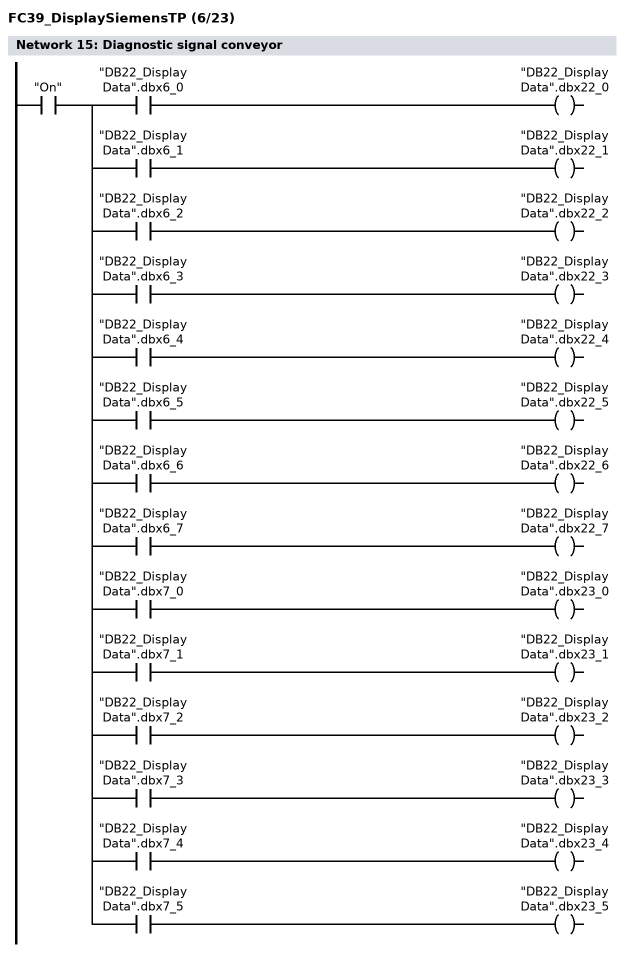
   RUNG wire#powerrail
      Contact( "On" )
      wire#w1
      Contact( "DB22_DisplayData".dbx6_0 )
      Coil( "DB22_DisplayData".dbx22_0 )
   END_RUNG
   RUNG wire#w1
      Contact( "DB22_DisplayData".dbx6_1 )
      Coil( "DB22_DisplayData".dbx22_1 )
   END_RUNG
   RUNG wire#w1
      Contact( "DB22_DisplayData".dbx6_2 )
      Coil( "DB22_DisplayData".dbx22_2 )
   END_RUNG
   RUNG wire#w1
      Contact( "DB22_DisplayData".dbx6_3 )
      Coil( "DB22_DisplayData".dbx22_3 )
   END_RUNG
   RUNG wire#w1
      Contact( "DB22_DisplayData".dbx6_4 )
      Coil( "DB22_DisplayData".dbx22_4 )
   END_RUNG
   RUNG wire#w1
      Contact( "DB22_DisplayData".dbx6_5 )
      Coil( "DB22_DisplayData".dbx22_5 )
   END_RUNG
   RUNG wire#w1
      Contact( "DB22_DisplayData".dbx6_6 )
      Coil( "DB22_DisplayData".dbx22_6 )
   END_RUNG
   RUNG wire#w1
      Contact( "DB22_DisplayData".dbx6_7 )
      Coil( "DB22_DisplayData".dbx22_7 )
   END_RUNG
   RUNG wire#w1
      Contact( "DB22_DisplayData".dbx7_0 )
      Coil( "DB22_DisplayData".dbx23_0 )
   END_RUNG
   RUNG wire#w1
      Contact( "DB22_DisplayData".dbx7_1 )
      Coil( "DB22_DisplayData".dbx23_1 )
   END_RUNG
   RUNG wire#w1
      Contact( "DB22_DisplayData".dbx7_2 )
      Coil( "DB22_DisplayData".dbx23_2 )
   END_RUNG
   RUNG wire#w1
      Contact( "DB22_DisplayData".dbx7_3 )
      Coil( "DB22_DisplayData".dbx23_3 )
   END_RUNG
   RUNG wire#w1
      Contact( "DB22_DisplayData".dbx7_4 )
      Coil( "DB22_DisplayData".dbx23_4 )
   END_RUNG
   RUNG wire#w1
      Contact( "DB22_DisplayData".dbx7_5 )
      Coil( "DB22_DisplayData".dbx23_5 )
   END_RUNG
   // the same network as SCL:
   "DB22_DisplayData".dbx22_0 := "On" AND "DB22_DisplayData".dbx6_0;
   "DB22_DisplayData".dbx22_1 := "On" AND "DB22_DisplayData".dbx6_1;
   "DB22_DisplayData".dbx22_2 := "On" AND "DB22_DisplayData".dbx6_2;
   "DB22_DisplayData".dbx22_3 := "On" AND "DB22_DisplayData".dbx6_3;
   "DB22_DisplayData".dbx22_4 := "On" AND "DB22_DisplayData".dbx6_4;
   "DB22_DisplayData".dbx22_5 := "On" AND "DB22_DisplayData".dbx6_5;
   "DB22_DisplayData".dbx22_6 := "On" AND "DB22_DisplayData".dbx6_6;
   "DB22_DisplayData".dbx22_7 := "On" AND "DB22_DisplayData".dbx6_7;
   "DB22_DisplayData".dbx23_0 := "On" AND "DB22_DisplayData".dbx7_0;
   "DB22_DisplayData".dbx23_1 := "On" AND "DB22_DisplayData".dbx7_1;
   "DB22_DisplayData".dbx23_2 := "On" AND "DB22_DisplayData".dbx7_2;
   "DB22_DisplayData".dbx23_3 := "On" AND "DB22_DisplayData".dbx7_3;
   "DB22_DisplayData".dbx23_4 := "On" AND "DB22_DisplayData".dbx7_4;
   "DB22_DisplayData".dbx23_5 := "On" AND "DB22_DisplayData".dbx7_5;
END_REGION

REGION Network 16: Diagnostic signal conveyor
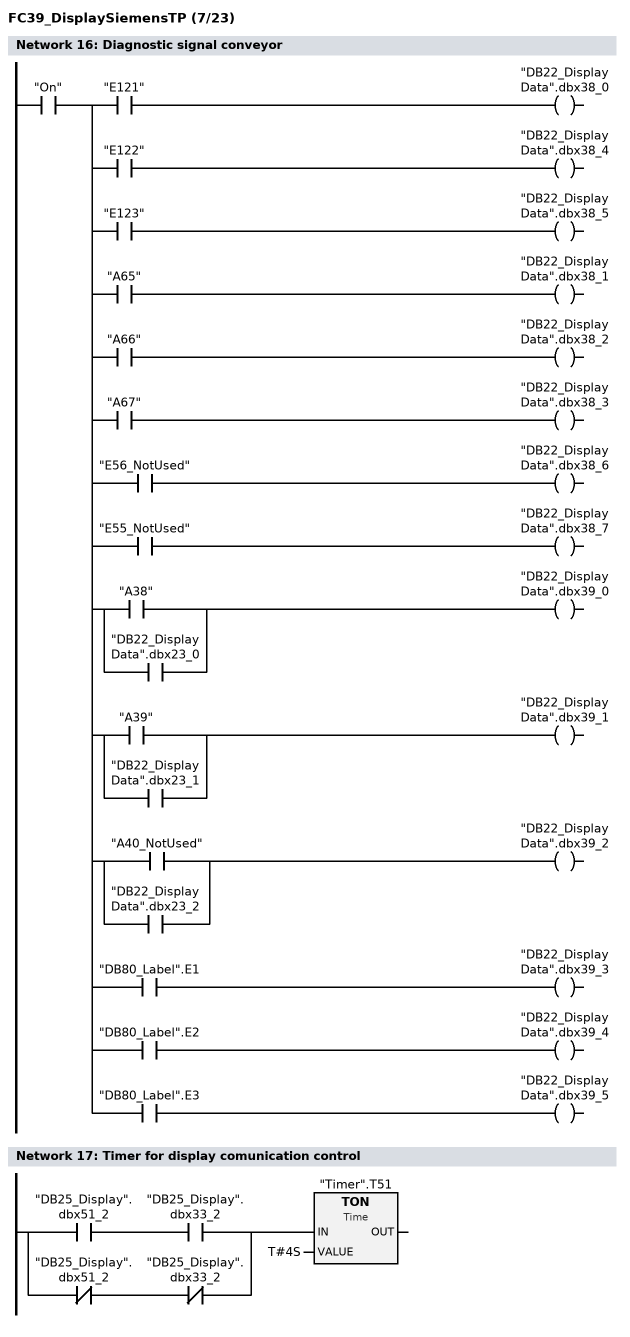
   RUNG wire#powerrail
      Contact( "On" )
      wire#w1
      Contact( "E121" )
      Coil( "DB22_DisplayData".dbx38_0 )
   END_RUNG
   RUNG wire#w1
      Contact( "E122" )
      Coil( "DB22_DisplayData".dbx38_4 )
   END_RUNG
   RUNG wire#w1
      Contact( "E123" )
      Coil( "DB22_DisplayData".dbx38_5 )
   END_RUNG
   RUNG wire#w1
      Contact( "A65" )
      Coil( "DB22_DisplayData".dbx38_1 )
   END_RUNG
   RUNG wire#w1
      Contact( "A66" )
      Coil( "DB22_DisplayData".dbx38_2 )
   END_RUNG
   RUNG wire#w1
      Contact( "A67" )
      Coil( "DB22_DisplayData".dbx38_3 )
   END_RUNG
   RUNG wire#w1
      Contact( "E56_NotUsed" )
      Coil( "DB22_DisplayData".dbx38_6 )
   END_RUNG
   RUNG wire#w1
      Contact( "E55_NotUsed" )
      Coil( "DB22_DisplayData".dbx38_7 )
   END_RUNG
   RUNG wire#w1
      Contact( "A38" )
      wire#w2
      Coil( "DB22_DisplayData".dbx39_0 )
   END_RUNG
   RUNG wire#w1
      Contact( "DB22_DisplayData".dbx23_0 )
   END_RUNG wire#w2
   RUNG wire#w1
      Contact( "A39" )
      wire#w3
      Coil( "DB22_DisplayData".dbx39_1 )
   END_RUNG
   RUNG wire#w1
      Contact( "DB22_DisplayData".dbx23_1 )
   END_RUNG wire#w3
   RUNG wire#w1
      Contact( "A40_NotUsed" )
      wire#w4
      Coil( "DB22_DisplayData".dbx39_2 )
   END_RUNG
   RUNG wire#w1
      Contact( "DB22_DisplayData".dbx23_2 )
   END_RUNG wire#w4
   RUNG wire#w1
      Contact( "DB80_Label".E1 )
      Coil( "DB22_DisplayData".dbx39_3 )
   END_RUNG
   RUNG wire#w1
      Contact( "DB80_Label".E2 )
      Coil( "DB22_DisplayData".dbx39_4 )
   END_RUNG
   RUNG wire#w1
      Contact( "DB80_Label".E3 )
      Coil( "DB22_DisplayData".dbx39_5 )
   END_RUNG
   // the same network as SCL:
   "DB22_DisplayData".dbx38_0 := "On" AND "E121";
   "DB22_DisplayData".dbx38_4 := "On" AND "E122";
   "DB22_DisplayData".dbx38_5 := "On" AND "E123";
   "DB22_DisplayData".dbx38_1 := "On" AND "A65";
   "DB22_DisplayData".dbx38_2 := "On" AND "A66";
   "DB22_DisplayData".dbx38_3 := "On" AND "A67";
   "DB22_DisplayData".dbx38_6 := "On" AND "E56_NotUsed";
   "DB22_DisplayData".dbx38_7 := "On" AND "E55_NotUsed";
   "DB22_DisplayData".dbx39_0 := "On" AND ("A38" OR "DB22_DisplayData".dbx23_0);
   "DB22_DisplayData".dbx39_1 := "On" AND ("A39" OR "DB22_DisplayData".dbx23_1);
   "DB22_DisplayData".dbx39_2 := "On" AND ("A40_NotUsed" OR "DB22_DisplayData".dbx23_2);
   "DB22_DisplayData".dbx39_3 := "On" AND "DB80_Label".E1;
   "DB22_DisplayData".dbx39_4 := "On" AND "DB80_Label".E2;
   "DB22_DisplayData".dbx39_5 := "On" AND "DB80_Label".E3;
END_REGION

REGION Network 17: Timer for display comunication control
   "Timer".T51.TON(IN := ("DB25_Display".dbx51_2 AND "DB25_Display".dbx33_2) OR (NOT "DB25_Display".dbx51_2 AND NOT "DB25_Display".dbx33_2), PT := T#4S);   // TON coil
END_REGION

REGION Network 18: Support for display communication timeout
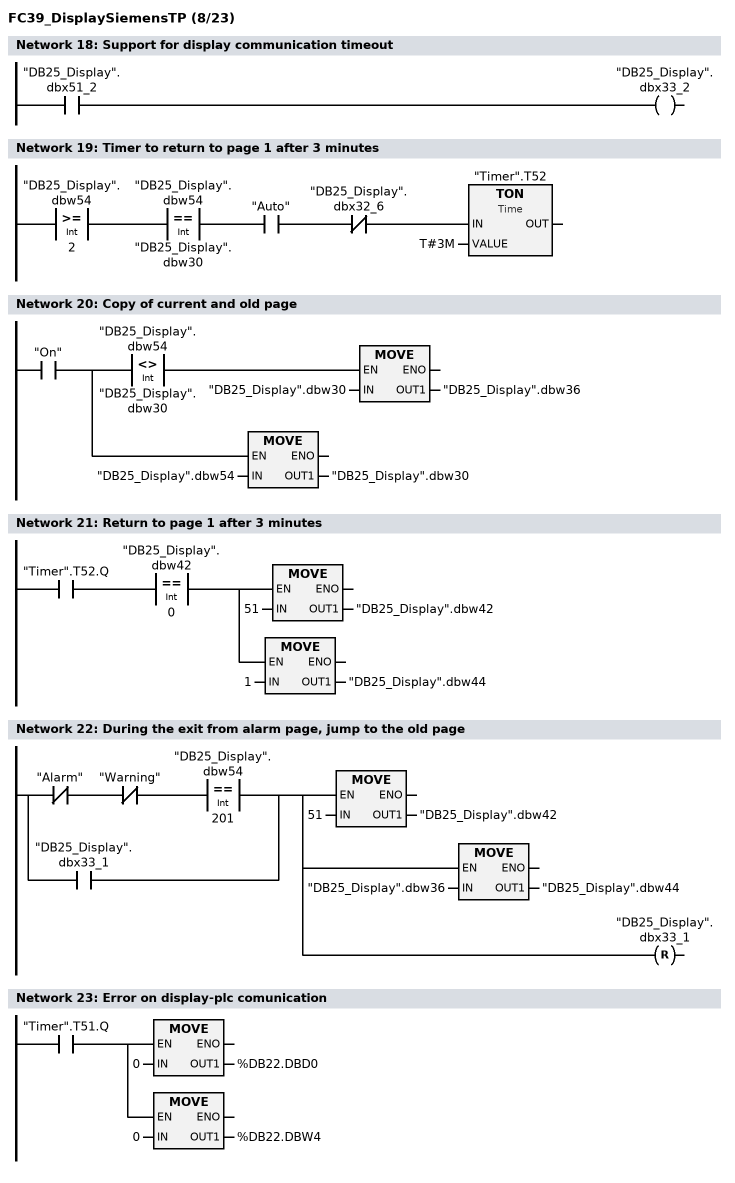
   RUNG wire#powerrail
      Contact( "DB25_Display".dbx51_2 )
      Coil( "DB25_Display".dbx33_2 )
   END_RUNG
   // the same network as SCL:
   "DB25_Display".dbx33_2 := "DB25_Display".dbx51_2;
END_REGION

REGION Network 19: Timer to return to page 1 after 3 minutes
   "Timer".T52.TON(IN := ("DB25_Display".dbw54 >= 2) AND ("DB25_Display".dbw54 = "DB25_Display".dbw30) AND "Auto" AND NOT "DB25_Display".dbx32_6, PT := T#3M);   // TON coil
END_REGION

REGION Network 20: Copy of current and old page
   RUNG wire#powerrail
      Contact( "On" )
      wire#w1
      { S7_Templates := "SrcType := Int" } NE_Contact(in1 := "DB25_Display".dbw54, in2 := "DB25_Display".dbw30)
      { S7_GenerateENO := "TRUE" } Move(in := "DB25_Display".dbw30, out1 => "DB25_Display".dbw36)
   END_RUNG
   RUNG wire#w1
      { S7_GenerateENO := "TRUE" } Move(in := "DB25_Display".dbw54, out1 => "DB25_Display".dbw30)
   END_RUNG
   // the same network as SCL:
   IF "On" AND ("DB25_Display".dbw54 <> "DB25_Display".dbw30) THEN
       "DB25_Display".dbw36 := "DB25_Display".dbw30;
   END_IF;
   IF "On" THEN "DB25_Display".dbw30 := "DB25_Display".dbw54; END_IF;
END_REGION

REGION Network 21: Return to page 1 after 3 minutes
   RUNG wire#powerrail
      Contact( "Timer".T52.Q )
      { S7_Templates := "SrcType := Int" } EQ_Contact(in1 := "DB25_Display".dbw42, in2 := 0)
      wire#w1
      { S7_GenerateENO := "TRUE" } Move(in := 51, out1 => "DB25_Display".dbw42)
   END_RUNG
   RUNG wire#w1
      { S7_GenerateENO := "TRUE" } Move(in := 1, out1 => "DB25_Display".dbw44)
   END_RUNG
   // the same network as SCL:
   #_w1 := "Timer".T52.Q AND ("DB25_Display".dbw42 = 0);
   IF #_w1 THEN
       "DB25_Display".dbw42 := 51;
       "DB25_Display".dbw44 := 1;
   END_IF;
END_REGION

REGION Network 22: During the exit from alarm page, jump to the old page
   RUNG wire#powerrail
      I_Contact( "Alarm" )
      I_Contact( "Warning" )
      { S7_Templates := "SrcType := Int" } EQ_Contact(in1 := "DB25_Display".dbw54, in2 := 201)
      wire#w1
      { S7_GenerateENO := "TRUE" } Move(in := 51, out1 => "DB25_Display".dbw42)
   END_RUNG
   RUNG wire#powerrail
      Contact( "DB25_Display".dbx33_1 )
   END_RUNG wire#w1
   RUNG wire#w1
      { S7_GenerateENO := "TRUE" } Move(in := "DB25_Display".dbw36, out1 => "DB25_Display".dbw44)
   END_RUNG
   RUNG wire#w1
      R_Coil( "DB25_Display".dbx33_1 )
   END_RUNG
   // the same network as SCL:
   IF (NOT "Alarm" AND NOT "Warning" AND ("DB25_Display".dbw54 = 201)) OR "DB25_Display".dbx33_1 THEN
       "DB25_Display".dbw42 := 51;
       "DB25_Display".dbw44 := "DB25_Display".dbw36;
       "DB25_Display".dbx33_1 := FALSE;
   END_IF;
END_REGION

REGION Network 23: Error on display-plc comunication
   RUNG wire#powerrail
      Contact( "Timer".T51.Q )
      wire#w1
      { S7_GenerateENO := "TRUE" } Move(in := 0, out1 => %DB22.DBD0)
   END_RUNG
   RUNG wire#w1
      { S7_GenerateENO := "TRUE" } Move(in := 0, out1 => %DB22.DBW4)
   END_RUNG
   // the same network as SCL:
   IF "Timer".T51.Q THEN
       %DB22.DBD0 := 0;
       %DB22.DBW4 := 0;
   END_IF;
END_REGION

REGION Network 24: Machine mode on Display
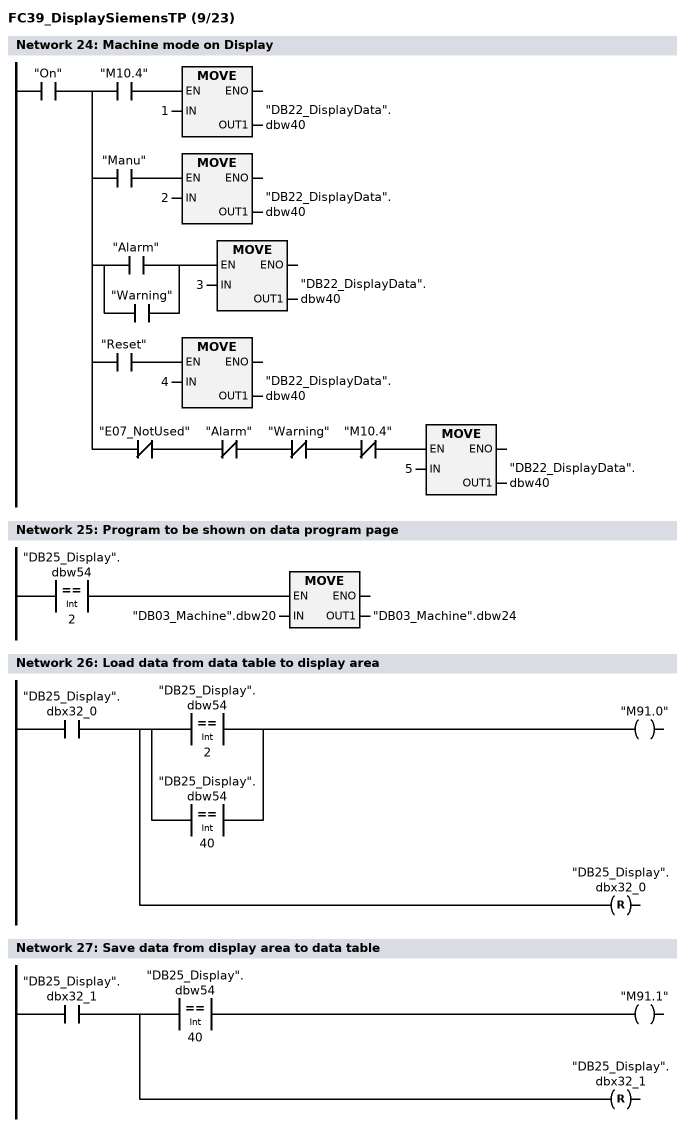
   RUNG wire#powerrail
      Contact( "On" )
      wire#w1
      Contact( "M10.4" )
      { S7_GenerateENO := "TRUE" } Move(in := 1, out1 => "DB22_DisplayData".dbw40)
   END_RUNG
   RUNG wire#w1
      Contact( "Manu" )
      { S7_GenerateENO := "TRUE" } Move(in := 2, out1 => "DB22_DisplayData".dbw40)
   END_RUNG
   RUNG wire#w1
      Contact( "Alarm" )
      wire#w2
      { S7_GenerateENO := "TRUE" } Move(in := 3, out1 => "DB22_DisplayData".dbw40)
   END_RUNG
   RUNG wire#w1
      Contact( "Warning" )
   END_RUNG wire#w2
   RUNG wire#w1
      Contact( "Reset" )
      { S7_GenerateENO := "TRUE" } Move(in := 4, out1 => "DB22_DisplayData".dbw40)
   END_RUNG
   RUNG wire#w1
      I_Contact( "E07_NotUsed" )
      I_Contact( "Alarm" )
      I_Contact( "Warning" )
      I_Contact( "M10.4" )
      { S7_GenerateENO := "TRUE" } Move(in := 5, out1 => "DB22_DisplayData".dbw40)
   END_RUNG
   // the same network as SCL:
   IF "On" AND "M10.4" THEN "DB22_DisplayData".dbw40 := 1; END_IF;
   IF "On" AND "Manu" THEN "DB22_DisplayData".dbw40 := 2; END_IF;
   IF "On" AND ("Alarm" OR "Warning") THEN "DB22_DisplayData".dbw40 := 3; END_IF;
   IF "On" AND "Reset" THEN "DB22_DisplayData".dbw40 := 4; END_IF;
   IF "On" AND NOT "E07_NotUsed" AND NOT "Alarm" AND NOT "Warning" AND NOT "M10.4" THEN
       "DB22_DisplayData".dbw40 := 5;
   END_IF;
END_REGION

REGION Network 25: Program to be shown on data program page
   RUNG wire#powerrail
      { S7_Templates := "SrcType := Int" } EQ_Contact(in1 := "DB25_Display".dbw54, in2 := 2)
      { S7_GenerateENO := "TRUE" } Move(in := "DB03_Machine".dbw20, out1 => "DB03_Machine".dbw24)
   END_RUNG
   // the same network as SCL:
   IF "DB25_Display".dbw54 = 2 THEN "DB03_Machine".dbw24 := "DB03_Machine".dbw20; END_IF;
END_REGION

REGION Network 26: Load data from data table to display area
   RUNG wire#powerrail
      Contact( "DB25_Display".dbx32_0 )
      wire#w1
      { S7_Templates := "SrcType := Int" } EQ_Contact(in1 := "DB25_Display".dbw54, in2 := 2)
      wire#w2
      Coil( "M91.0" )
   END_RUNG
   RUNG wire#w1
      { S7_Templates := "SrcType := Int" } EQ_Contact(in1 := "DB25_Display".dbw54, in2 := 40)
   END_RUNG wire#w2
   RUNG wire#w1
      R_Coil( "DB25_Display".dbx32_0 )
   END_RUNG
   // the same network as SCL:
   "M91.0" := "DB25_Display".dbx32_0 AND (("DB25_Display".dbw54 = 2) OR ("DB25_Display".dbw54 = 40));
   IF "DB25_Display".dbx32_0 THEN "DB25_Display".dbx32_0 := FALSE; END_IF;
END_REGION

REGION Network 27: Save data from display area to data table
   RUNG wire#powerrail
      Contact( "DB25_Display".dbx32_1 )
      wire#w1
      { S7_Templates := "SrcType := Int" } EQ_Contact(in1 := "DB25_Display".dbw54, in2 := 40)
      Coil( "M91.1" )
   END_RUNG
   RUNG wire#w1
      R_Coil( "DB25_Display".dbx32_1 )
   END_RUNG
   // the same network as SCL:
   "M91.1" := "DB25_Display".dbx32_1 AND ("DB25_Display".dbw54 = 40);
   IF "DB25_Display".dbx32_1 THEN "DB25_Display".dbx32_1 := FALSE; END_IF;
END_REGION

REGION Network 28: Program bit: Blink load button
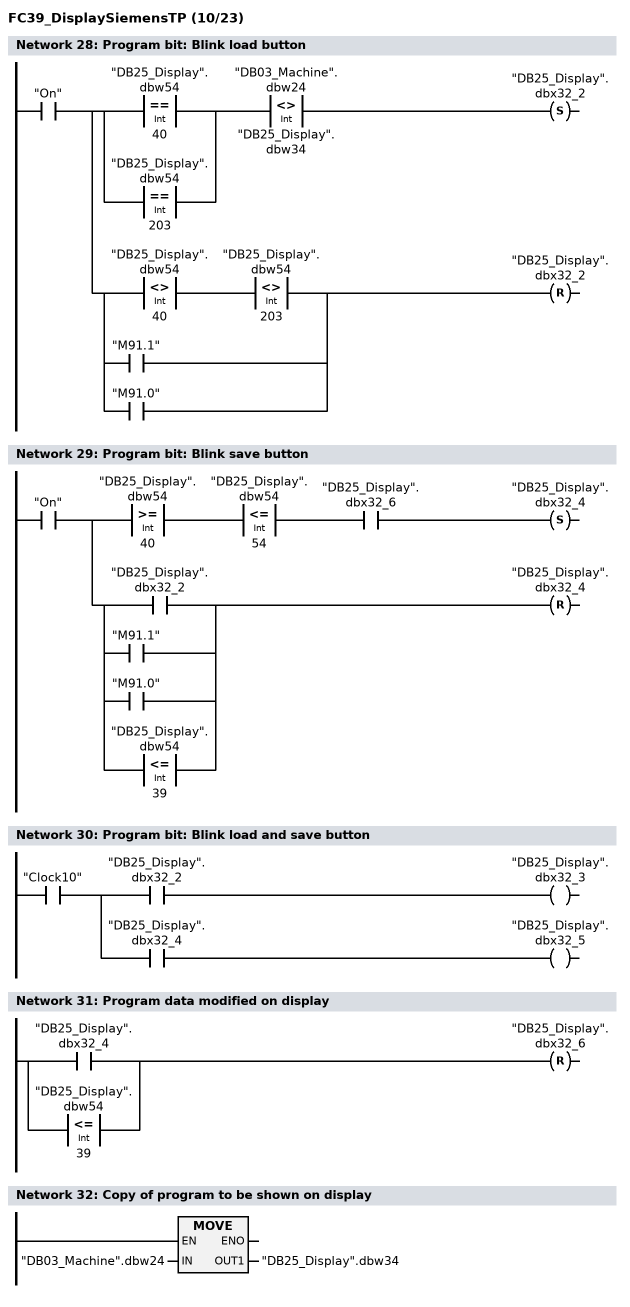
   RUNG wire#powerrail
      Contact( "On" )
      wire#w1
      { S7_Templates := "SrcType := Int" } EQ_Contact(in1 := "DB25_Display".dbw54, in2 := 40)
      wire#w2
      { S7_Templates := "SrcType := Int" } NE_Contact(in1 := "DB03_Machine".dbw24, in2 := "DB25_Display".dbw34)
      S_Coil( "DB25_Display".dbx32_2 )
   END_RUNG
   RUNG wire#w1
      { S7_Templates := "SrcType := Int" } EQ_Contact(in1 := "DB25_Display".dbw54, in2 := 203)
   END_RUNG wire#w2
   RUNG wire#w1
      { S7_Templates := "SrcType := Int" } NE_Contact(in1 := "DB25_Display".dbw54, in2 := 40)
      { S7_Templates := "SrcType := Int" } NE_Contact(in1 := "DB25_Display".dbw54, in2 := 203)
      wire#w3
      R_Coil( "DB25_Display".dbx32_2 )
   END_RUNG
   RUNG wire#w1
      Contact( "M91.1" )
   END_RUNG wire#w3
   RUNG wire#w1
      Contact( "M91.0" )
   END_RUNG wire#w3
   // the same network as SCL:
   IF "On" AND (("DB25_Display".dbw54 = 40) OR ("DB25_Display".dbw54 = 203)) AND ("DB03_Machine".dbw24 <> "DB25_Display".dbw34) THEN
       "DB25_Display".dbx32_2 := TRUE;
   END_IF;
   IF "On" AND ((("DB25_Display".dbw54 <> 40) AND ("DB25_Display".dbw54 <> 203)) OR "M91.1" OR "M91.0") THEN
       "DB25_Display".dbx32_2 := FALSE;
   END_IF;
END_REGION

REGION Network 29: Program bit: Blink save button
   RUNG wire#powerrail
      Contact( "On" )
      wire#w1
      { S7_Templates := "SrcType := Int" } GE_Contact(in1 := "DB25_Display".dbw54, in2 := 40)
      { S7_Templates := "SrcType := Int" } LE_Contact(in1 := "DB25_Display".dbw54, in2 := 54)
      Contact( "DB25_Display".dbx32_6 )
      S_Coil( "DB25_Display".dbx32_4 )
   END_RUNG
   RUNG wire#w1
      Contact( "DB25_Display".dbx32_2 )
      wire#w2
      R_Coil( "DB25_Display".dbx32_4 )
   END_RUNG
   RUNG wire#w1
      Contact( "M91.1" )
   END_RUNG wire#w2
   RUNG wire#w1
      Contact( "M91.0" )
   END_RUNG wire#w2
   RUNG wire#w1
      { S7_Templates := "SrcType := Int" } LE_Contact(in1 := "DB25_Display".dbw54, in2 := 39)
   END_RUNG wire#w2
   // the same network as SCL:
   IF "On" AND ("DB25_Display".dbw54 >= 40) AND ("DB25_Display".dbw54 <= 54) AND "DB25_Display".dbx32_6 THEN
       "DB25_Display".dbx32_4 := TRUE;
   END_IF;
   IF "On" AND ("DB25_Display".dbx32_2 OR "M91.1" OR "M91.0" OR ("DB25_Display".dbw54 <= 39)) THEN
       "DB25_Display".dbx32_4 := FALSE;
   END_IF;
END_REGION

REGION Network 30: Program bit: Blink load and save button
   RUNG wire#powerrail
      Contact( "Clock10" )
      wire#w1
      Contact( "DB25_Display".dbx32_2 )
      Coil( "DB25_Display".dbx32_3 )
   END_RUNG
   RUNG wire#w1
      Contact( "DB25_Display".dbx32_4 )
      Coil( "DB25_Display".dbx32_5 )
   END_RUNG
   // the same network as SCL:
   "DB25_Display".dbx32_3 := "Clock10" AND "DB25_Display".dbx32_2;
   "DB25_Display".dbx32_5 := "Clock10" AND "DB25_Display".dbx32_4;
END_REGION

REGION Network 31: Program data modified on display
   RUNG wire#powerrail
      Contact( "DB25_Display".dbx32_4 )
      wire#w1
      R_Coil( "DB25_Display".dbx32_6 )
   END_RUNG
   RUNG wire#powerrail
      { S7_Templates := "SrcType := Int" } LE_Contact(in1 := "DB25_Display".dbw54, in2 := 39)
   END_RUNG wire#w1
   // the same network as SCL:
   IF "DB25_Display".dbx32_4 OR ("DB25_Display".dbw54 <= 39) THEN "DB25_Display".dbx32_6 := FALSE; END_IF;
END_REGION

REGION Network 32: Copy of program to be shown on display
   RUNG wire#powerrail
      { S7_GenerateENO := "TRUE" } Move(in := "DB03_Machine".dbw24, out1 => "DB25_Display".dbw34)
   END_RUNG
   // the same network as SCL:
   "DB25_Display".dbw34 := "DB03_Machine".dbw24;
END_REGION

REGION Network 33: Grey bar data: Active program
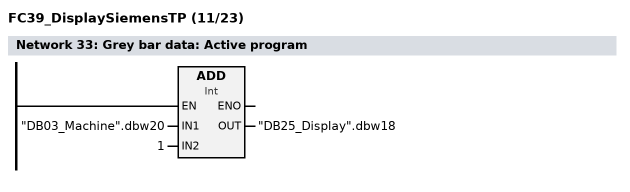
   RUNG wire#powerrail
      { S7_Templates := "SrcType := Int"; S7_GenerateENO := "TRUE" } Add(in1 := "DB03_Machine".dbw20, in2 := 1, out => "DB25_Display".dbw18)
   END_RUNG
   // the same network as SCL:
   "DB25_Display".dbw18 := "DB03_Machine".dbw20 + 1;
END_REGION

REGION Network 35: Support memory for pressure plate grey bar
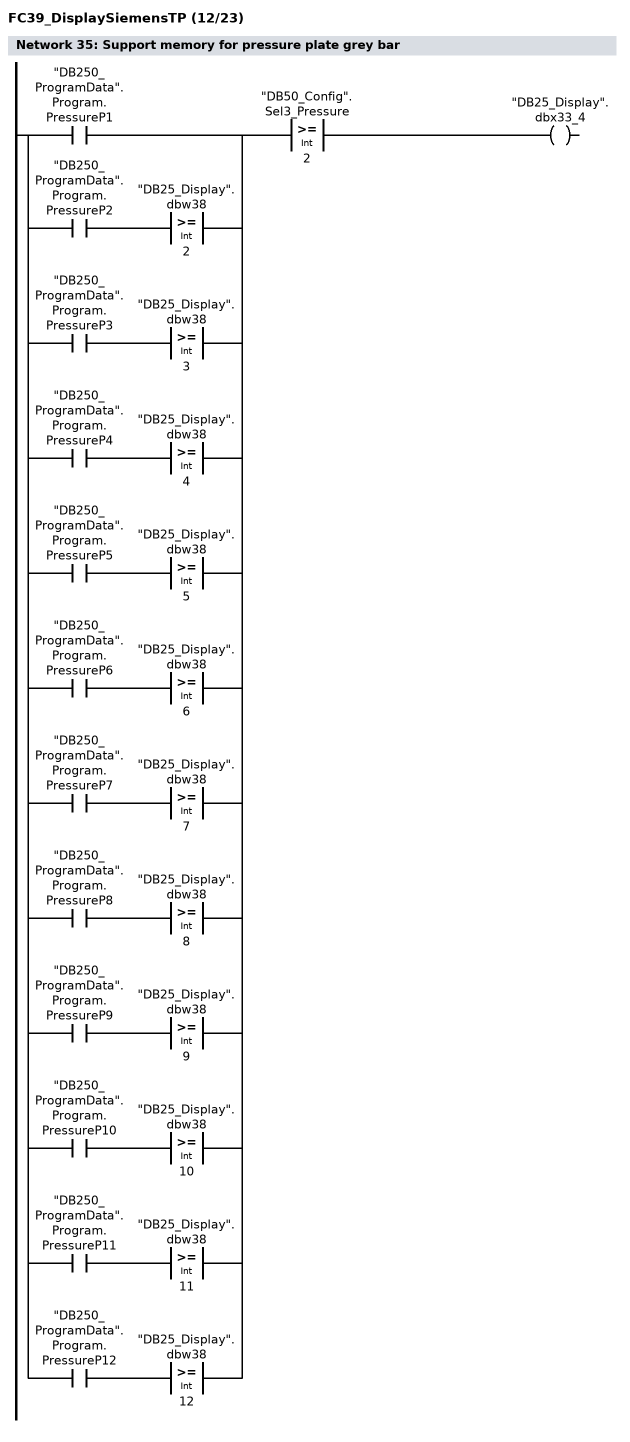
   RUNG wire#powerrail
      Contact( "DB250_ProgramData".Program.PressureP1 )
      wire#w1
      { S7_Templates := "SrcType := Int" } GE_Contact(in1 := "DB50_Config".Sel3_Pressure, in2 := 2)
      Coil( "DB25_Display".dbx33_4 )
   END_RUNG
   RUNG wire#powerrail
      Contact( "DB250_ProgramData".Program.PressureP2 )
      { S7_Templates := "SrcType := Int" } GE_Contact(in1 := "DB25_Display".dbw38, in2 := 2)
   END_RUNG wire#w1
   RUNG wire#powerrail
      Contact( "DB250_ProgramData".Program.PressureP3 )
      { S7_Templates := "SrcType := Int" } GE_Contact(in1 := "DB25_Display".dbw38, in2 := 3)
   END_RUNG wire#w1
   RUNG wire#powerrail
      Contact( "DB250_ProgramData".Program.PressureP4 )
      { S7_Templates := "SrcType := Int" } GE_Contact(in1 := "DB25_Display".dbw38, in2 := 4)
   END_RUNG wire#w1
   RUNG wire#powerrail
      Contact( "DB250_ProgramData".Program.PressureP5 )
      { S7_Templates := "SrcType := Int" } GE_Contact(in1 := "DB25_Display".dbw38, in2 := 5)
   END_RUNG wire#w1
   RUNG wire#powerrail
      Contact( "DB250_ProgramData".Program.PressureP6 )
      { S7_Templates := "SrcType := Int" } GE_Contact(in1 := "DB25_Display".dbw38, in2 := 6)
   END_RUNG wire#w1
   RUNG wire#powerrail
      Contact( "DB250_ProgramData".Program.PressureP7 )
      { S7_Templates := "SrcType := Int" } GE_Contact(in1 := "DB25_Display".dbw38, in2 := 7)
   END_RUNG wire#w1
   RUNG wire#powerrail
      Contact( "DB250_ProgramData".Program.PressureP8 )
      { S7_Templates := "SrcType := Int" } GE_Contact(in1 := "DB25_Display".dbw38, in2 := 8)
   END_RUNG wire#w1
   RUNG wire#powerrail
      Contact( "DB250_ProgramData".Program.PressureP9 )
      { S7_Templates := "SrcType := Int" } GE_Contact(in1 := "DB25_Display".dbw38, in2 := 9)
   END_RUNG wire#w1
   RUNG wire#powerrail
      Contact( "DB250_ProgramData".Program.PressureP10 )
      { S7_Templates := "SrcType := Int" } GE_Contact(in1 := "DB25_Display".dbw38, in2 := 10)
   END_RUNG wire#w1
   RUNG wire#powerrail
      Contact( "DB250_ProgramData".Program.PressureP11 )
      { S7_Templates := "SrcType := Int" } GE_Contact(in1 := "DB25_Display".dbw38, in2 := 11)
   END_RUNG wire#w1
   RUNG wire#powerrail
      Contact( "DB250_ProgramData".Program.PressureP12 )
      { S7_Templates := "SrcType := Int" } GE_Contact(in1 := "DB25_Display".dbw38, in2 := 12)
   END_RUNG wire#w1
   // the same network as SCL:
   "DB25_Display".dbx33_4 := ("DB250_ProgramData".Program.PressureP1 OR ("DB250_ProgramData".Program.PressureP2 AND ("DB25_Display".dbw38 >= 2)) OR ("DB250_ProgramData".Program.PressureP3 AND ("DB25_Display".dbw38 >= 3)) OR ("DB250_ProgramData".Program.PressureP4 AND ("DB25_Display".dbw38 >= 4)) OR ("DB250_ProgramData".Program.PressureP5 AND ("DB25_Display".dbw38 >= 5)) OR ("DB250_ProgramData".Program.PressureP6 AND ("DB25_Display".dbw38 >= 6)) OR ("DB250_ProgramData".Program.PressureP7 AND ("DB25_Display".dbw38 >= 7)) OR ("DB250_ProgramData".Program.PressureP8 AND ("DB25_Display".dbw38 >= 8)) OR ("DB250_ProgramData".Program.PressureP9 AND ("DB25_Display".dbw38 >= 9)) OR ("DB250_ProgramData".Program.PressureP10 AND ("DB25_Display".dbw38 >= 10)) OR ("DB250_ProgramData".Program.PressureP11 AND ("DB25_Display".dbw38 >= 11)) OR ("DB250_ProgramData".Program.PressureP12 AND ("DB25_Display".dbw38 >= 12))) AND ("DB50_Config".Sel3_Pressure >= 2);
END_REGION

REGION Network 36: Support memory for lifter grey bar
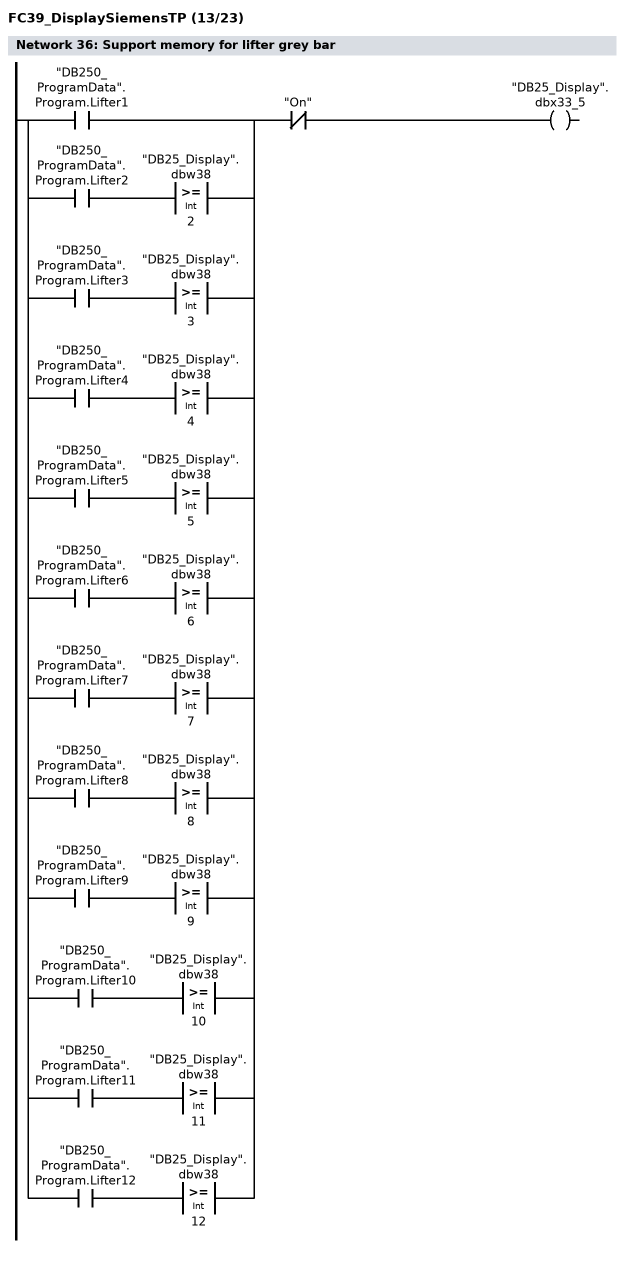
   RUNG wire#powerrail
      Contact( "DB250_ProgramData".Program.Lifter1 )
      wire#w1
      I_Contact( "On" )
      Coil( "DB25_Display".dbx33_5 )
   END_RUNG
   RUNG wire#powerrail
      Contact( "DB250_ProgramData".Program.Lifter2 )
      { S7_Templates := "SrcType := Int" } GE_Contact(in1 := "DB25_Display".dbw38, in2 := 2)
   END_RUNG wire#w1
   RUNG wire#powerrail
      Contact( "DB250_ProgramData".Program.Lifter3 )
      { S7_Templates := "SrcType := Int" } GE_Contact(in1 := "DB25_Display".dbw38, in2 := 3)
   END_RUNG wire#w1
   RUNG wire#powerrail
      Contact( "DB250_ProgramData".Program.Lifter4 )
      { S7_Templates := "SrcType := Int" } GE_Contact(in1 := "DB25_Display".dbw38, in2 := 4)
   END_RUNG wire#w1
   RUNG wire#powerrail
      Contact( "DB250_ProgramData".Program.Lifter5 )
      { S7_Templates := "SrcType := Int" } GE_Contact(in1 := "DB25_Display".dbw38, in2 := 5)
   END_RUNG wire#w1
   RUNG wire#powerrail
      Contact( "DB250_ProgramData".Program.Lifter6 )
      { S7_Templates := "SrcType := Int" } GE_Contact(in1 := "DB25_Display".dbw38, in2 := 6)
   END_RUNG wire#w1
   RUNG wire#powerrail
      Contact( "DB250_ProgramData".Program.Lifter7 )
      { S7_Templates := "SrcType := Int" } GE_Contact(in1 := "DB25_Display".dbw38, in2 := 7)
   END_RUNG wire#w1
   RUNG wire#powerrail
      Contact( "DB250_ProgramData".Program.Lifter8 )
      { S7_Templates := "SrcType := Int" } GE_Contact(in1 := "DB25_Display".dbw38, in2 := 8)
   END_RUNG wire#w1
   RUNG wire#powerrail
      Contact( "DB250_ProgramData".Program.Lifter9 )
      { S7_Templates := "SrcType := Int" } GE_Contact(in1 := "DB25_Display".dbw38, in2 := 9)
   END_RUNG wire#w1
   RUNG wire#powerrail
      Contact( "DB250_ProgramData".Program.Lifter10 )
      { S7_Templates := "SrcType := Int" } GE_Contact(in1 := "DB25_Display".dbw38, in2 := 10)
   END_RUNG wire#w1
   RUNG wire#powerrail
      Contact( "DB250_ProgramData".Program.Lifter11 )
      { S7_Templates := "SrcType := Int" } GE_Contact(in1 := "DB25_Display".dbw38, in2 := 11)
   END_RUNG wire#w1
   RUNG wire#powerrail
      Contact( "DB250_ProgramData".Program.Lifter12 )
      { S7_Templates := "SrcType := Int" } GE_Contact(in1 := "DB25_Display".dbw38, in2 := 12)
   END_RUNG wire#w1
   // the same network as SCL:
   "DB25_Display".dbx33_5 := ("DB250_ProgramData".Program.Lifter1 OR ("DB250_ProgramData".Program.Lifter2 AND ("DB25_Display".dbw38 >= 2)) OR ("DB250_ProgramData".Program.Lifter3 AND ("DB25_Display".dbw38 >= 3)) OR ("DB250_ProgramData".Program.Lifter4 AND ("DB25_Display".dbw38 >= 4)) OR ("DB250_ProgramData".Program.Lifter5 AND ("DB25_Display".dbw38 >= 5)) OR ("DB250_ProgramData".Program.Lifter6 AND ("DB25_Display".dbw38 >= 6)) OR ("DB250_ProgramData".Program.Lifter7 AND ("DB25_Display".dbw38 >= 7)) OR ("DB250_ProgramData".Program.Lifter8 AND ("DB25_Display".dbw38 >= 8)) OR ("DB250_ProgramData".Program.Lifter9 AND ("DB25_Display".dbw38 >= 9)) OR ("DB250_ProgramData".Program.Lifter10 AND ("DB25_Display".dbw38 >= 10)) OR ("DB250_ProgramData".Program.Lifter11 AND ("DB25_Display".dbw38 >= 11)) OR ("DB250_ProgramData".Program.Lifter12 AND ("DB25_Display".dbw38 >= 12))) AND NOT "On";
END_REGION

REGION Network 37: Grey bar data: Wrapping, Top, Pressure plate and Lifter
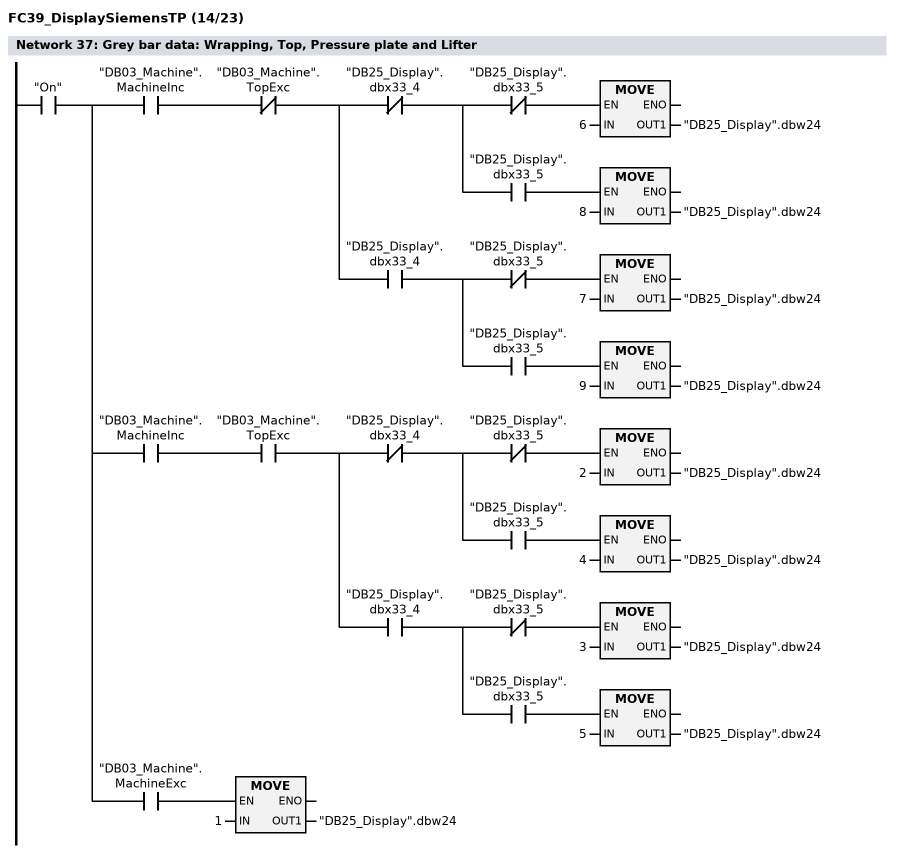
   RUNG wire#powerrail
      Contact( "On" )
      wire#w1
      Contact( "DB03_Machine".MachineInc )
      I_Contact( "DB03_Machine".TopExc )
      wire#w2
      I_Contact( "DB25_Display".dbx33_4 )
      wire#w3
      I_Contact( "DB25_Display".dbx33_5 )
      { S7_GenerateENO := "TRUE" } Move(in := 6, out1 => "DB25_Display".dbw24)
   END_RUNG
   RUNG wire#w3
      Contact( "DB25_Display".dbx33_5 )
      { S7_GenerateENO := "TRUE" } Move(in := 8, out1 => "DB25_Display".dbw24)
   END_RUNG
   RUNG wire#w2
      Contact( "DB25_Display".dbx33_4 )
      wire#w4
      I_Contact( "DB25_Display".dbx33_5 )
      { S7_GenerateENO := "TRUE" } Move(in := 7, out1 => "DB25_Display".dbw24)
   END_RUNG
   RUNG wire#w4
      Contact( "DB25_Display".dbx33_5 )
      { S7_GenerateENO := "TRUE" } Move(in := 9, out1 => "DB25_Display".dbw24)
   END_RUNG
   RUNG wire#w1
      Contact( "DB03_Machine".MachineInc )
      Contact( "DB03_Machine".TopExc )
      wire#w5
      I_Contact( "DB25_Display".dbx33_4 )
      wire#w6
      I_Contact( "DB25_Display".dbx33_5 )
      { S7_GenerateENO := "TRUE" } Move(in := 2, out1 => "DB25_Display".dbw24)
   END_RUNG
   RUNG wire#w6
      Contact( "DB25_Display".dbx33_5 )
      { S7_GenerateENO := "TRUE" } Move(in := 4, out1 => "DB25_Display".dbw24)
   END_RUNG
   RUNG wire#w5
      Contact( "DB25_Display".dbx33_4 )
      wire#w7
      I_Contact( "DB25_Display".dbx33_5 )
      { S7_GenerateENO := "TRUE" } Move(in := 3, out1 => "DB25_Display".dbw24)
   END_RUNG
   RUNG wire#w7
      Contact( "DB25_Display".dbx33_5 )
      { S7_GenerateENO := "TRUE" } Move(in := 5, out1 => "DB25_Display".dbw24)
   END_RUNG
   RUNG wire#w1
      Contact( "DB03_Machine".MachineExc )
      { S7_GenerateENO := "TRUE" } Move(in := 1, out1 => "DB25_Display".dbw24)
   END_RUNG
   // the same network as SCL:
   #_w1 := "On" AND "DB03_Machine".MachineInc AND NOT "DB03_Machine".TopExc;
   #_w2 := #_w1 AND NOT "DB25_Display".dbx33_4;
   IF #_w2 AND NOT "DB25_Display".dbx33_5 THEN "DB25_Display".dbw24 := 6; END_IF;
   IF #_w2 AND "DB25_Display".dbx33_5 THEN "DB25_Display".dbw24 := 8; END_IF;
   #_w3 := #_w1 AND "DB25_Display".dbx33_4;
   IF #_w3 AND NOT "DB25_Display".dbx33_5 THEN "DB25_Display".dbw24 := 7; END_IF;
   IF #_w3 AND "DB25_Display".dbx33_5 THEN "DB25_Display".dbw24 := 9; END_IF;
   #_w4 := "On" AND "DB03_Machine".MachineInc AND "DB03_Machine".TopExc;
   #_w5 := #_w4 AND NOT "DB25_Display".dbx33_4;
   IF #_w5 AND NOT "DB25_Display".dbx33_5 THEN "DB25_Display".dbw24 := 2; END_IF;
   IF #_w5 AND "DB25_Display".dbx33_5 THEN "DB25_Display".dbw24 := 4; END_IF;
   #_w6 := #_w4 AND "DB25_Display".dbx33_4;
   IF #_w6 AND NOT "DB25_Display".dbx33_5 THEN "DB25_Display".dbw24 := 3; END_IF;
   IF #_w6 AND "DB25_Display".dbx33_5 THEN "DB25_Display".dbw24 := 5; END_IF;
   IF "On" AND "DB03_Machine".MachineExc THEN "DB25_Display".dbw24 := 1; END_IF;
END_REGION

REGION Network 38: Grey bar data: Quote active
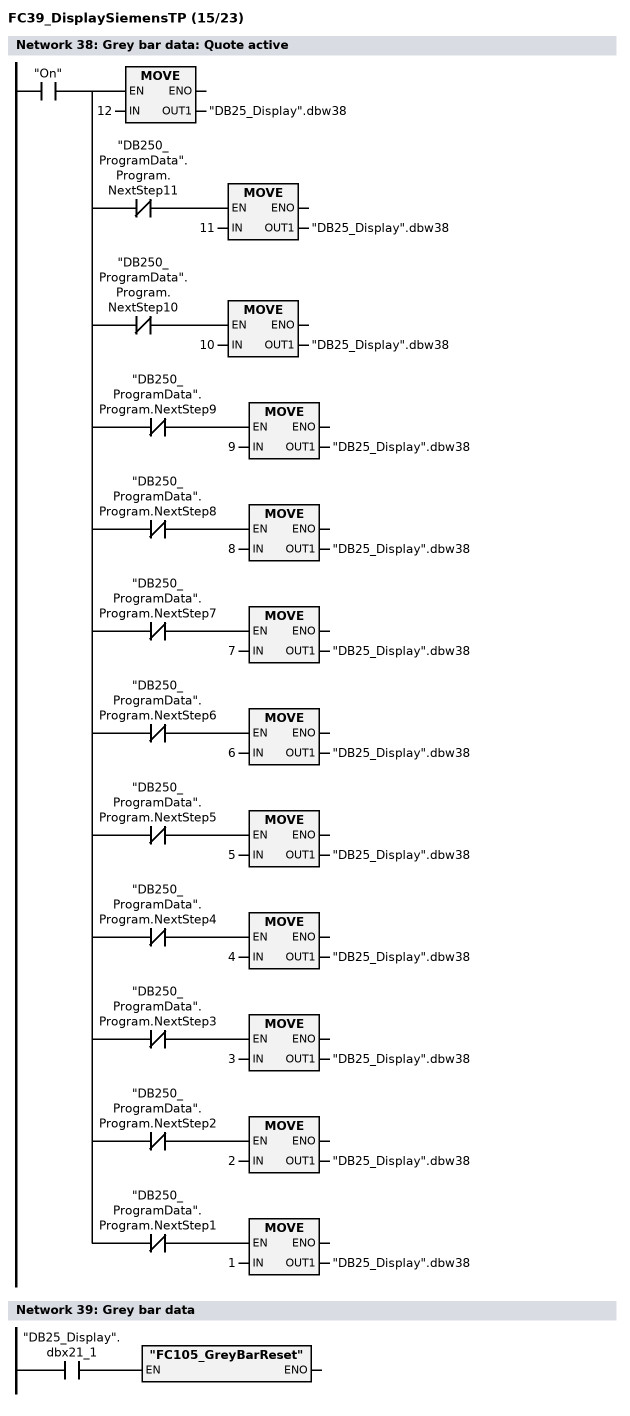
   RUNG wire#powerrail
      Contact( "On" )
      wire#w1
      { S7_GenerateENO := "TRUE" } Move(in := 12, out1 => "DB25_Display".dbw38)
   END_RUNG
   RUNG wire#w1
      I_Contact( "DB250_ProgramData".Program.NextStep11 )
      { S7_GenerateENO := "TRUE" } Move(in := 11, out1 => "DB25_Display".dbw38)
   END_RUNG
   RUNG wire#w1
      I_Contact( "DB250_ProgramData".Program.NextStep10 )
      { S7_GenerateENO := "TRUE" } Move(in := 10, out1 => "DB25_Display".dbw38)
   END_RUNG
   RUNG wire#w1
      I_Contact( "DB250_ProgramData".Program.NextStep9 )
      { S7_GenerateENO := "TRUE" } Move(in := 9, out1 => "DB25_Display".dbw38)
   END_RUNG
   RUNG wire#w1
      I_Contact( "DB250_ProgramData".Program.NextStep8 )
      { S7_GenerateENO := "TRUE" } Move(in := 8, out1 => "DB25_Display".dbw38)
   END_RUNG
   RUNG wire#w1
      I_Contact( "DB250_ProgramData".Program.NextStep7 )
      { S7_GenerateENO := "TRUE" } Move(in := 7, out1 => "DB25_Display".dbw38)
   END_RUNG
   RUNG wire#w1
      I_Contact( "DB250_ProgramData".Program.NextStep6 )
      { S7_GenerateENO := "TRUE" } Move(in := 6, out1 => "DB25_Display".dbw38)
   END_RUNG
   RUNG wire#w1
      I_Contact( "DB250_ProgramData".Program.NextStep5 )
      { S7_GenerateENO := "TRUE" } Move(in := 5, out1 => "DB25_Display".dbw38)
   END_RUNG
   RUNG wire#w1
      I_Contact( "DB250_ProgramData".Program.NextStep4 )
      { S7_GenerateENO := "TRUE" } Move(in := 4, out1 => "DB25_Display".dbw38)
   END_RUNG
   RUNG wire#w1
      I_Contact( "DB250_ProgramData".Program.NextStep3 )
      { S7_GenerateENO := "TRUE" } Move(in := 3, out1 => "DB25_Display".dbw38)
   END_RUNG
   RUNG wire#w1
      I_Contact( "DB250_ProgramData".Program.NextStep2 )
      { S7_GenerateENO := "TRUE" } Move(in := 2, out1 => "DB25_Display".dbw38)
   END_RUNG
   RUNG wire#w1
      I_Contact( "DB250_ProgramData".Program.NextStep1 )
      { S7_GenerateENO := "TRUE" } Move(in := 1, out1 => "DB25_Display".dbw38)
   END_RUNG
   // the same network as SCL:
   IF "On" THEN "DB25_Display".dbw38 := 12; END_IF;
   IF "On" AND NOT "DB250_ProgramData".Program.NextStep11 THEN "DB25_Display".dbw38 := 11; END_IF;
   IF "On" AND NOT "DB250_ProgramData".Program.NextStep10 THEN "DB25_Display".dbw38 := 10; END_IF;
   IF "On" AND NOT "DB250_ProgramData".Program.NextStep9 THEN "DB25_Display".dbw38 := 9; END_IF;
   IF "On" AND NOT "DB250_ProgramData".Program.NextStep8 THEN "DB25_Display".dbw38 := 8; END_IF;
   IF "On" AND NOT "DB250_ProgramData".Program.NextStep7 THEN "DB25_Display".dbw38 := 7; END_IF;
   IF "On" AND NOT "DB250_ProgramData".Program.NextStep6 THEN "DB25_Display".dbw38 := 6; END_IF;
   IF "On" AND NOT "DB250_ProgramData".Program.NextStep5 THEN "DB25_Display".dbw38 := 5; END_IF;
   IF "On" AND NOT "DB250_ProgramData".Program.NextStep4 THEN "DB25_Display".dbw38 := 4; END_IF;
   IF "On" AND NOT "DB250_ProgramData".Program.NextStep3 THEN "DB25_Display".dbw38 := 3; END_IF;
   IF "On" AND NOT "DB250_ProgramData".Program.NextStep2 THEN "DB25_Display".dbw38 := 2; END_IF;
   IF "On" AND NOT "DB250_ProgramData".Program.NextStep1 THEN "DB25_Display".dbw38 := 1; END_IF;
END_REGION

REGION Network 39: Grey bar data
   RUNG wire#powerrail
      Contact( "DB25_Display".dbx21_1 )
      "FC105_GreyBarReset"()
   END_RUNG
   // the same network as SCL:
   IF "DB25_Display".dbx21_1 THEN "FC105_GreyBarReset"(); END_IF;
END_REGION

REGION Network 40: Grey bar data
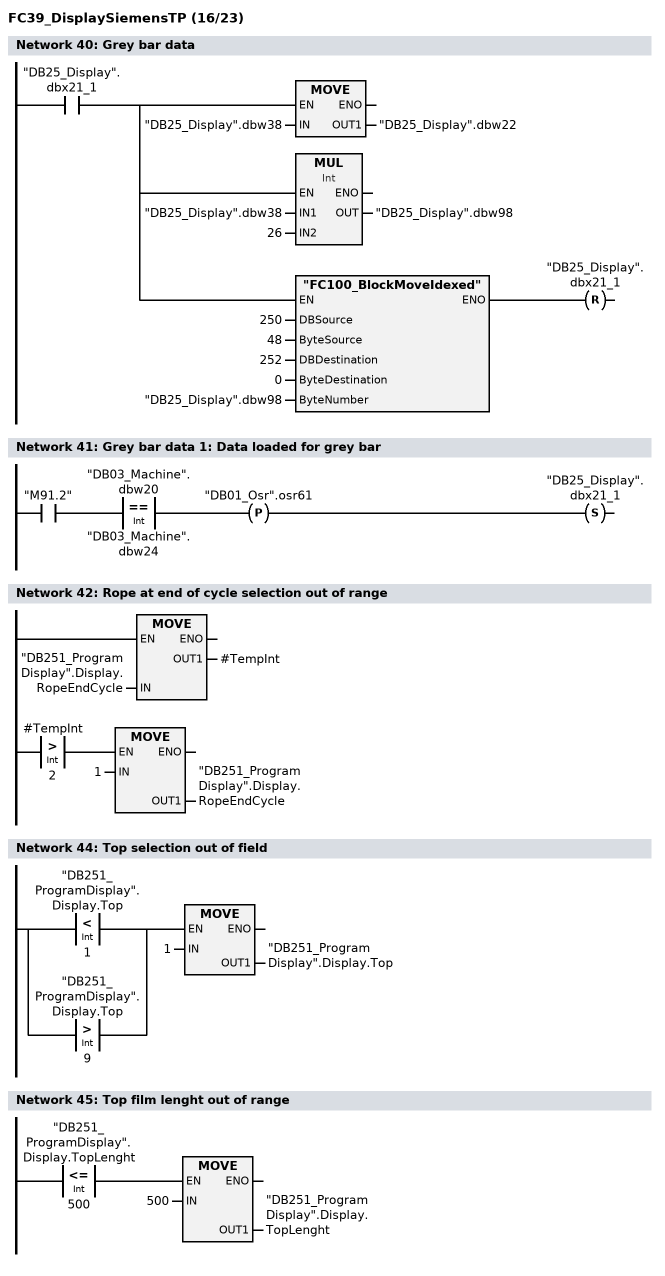
   RUNG wire#powerrail
      Contact( "DB25_Display".dbx21_1 )
      wire#w1
      { S7_GenerateENO := "TRUE" } Move(in := "DB25_Display".dbw38, out1 => "DB25_Display".dbw22)
   END_RUNG
   RUNG wire#w1
      { S7_Templates := "SrcType := Int"; S7_GenerateENO := "TRUE" } Mul(in1 := "DB25_Display".dbw38, in2 := 26, out => "DB25_Display".dbw98)
   END_RUNG
   RUNG wire#w1
      "FC100_BlockMoveIdexed"(DBSource := 250, ByteSource := 48, DBDestination := 252, ByteDestination := 0, ByteNumber := "DB25_Display".dbw98)
      R_Coil( "DB25_Display".dbx21_1 )
   END_RUNG
   // the same network as SCL:
   IF "DB25_Display".dbx21_1 THEN
       "DB25_Display".dbw22 := "DB25_Display".dbw38;
       "DB25_Display".dbw98 := "DB25_Display".dbw38 * 26;
   END_IF;
   "FC100_BlockMoveIdexed"(EN := "DB25_Display".dbx21_1,
                           DBSource := 250,
                           ByteSource := 48,
                           DBDestination := 252,
                           ByteDestination := 0,
                           ByteNumber := "DB25_Display".dbw98,
                           ENO => #_w1);
   IF #_w1 THEN "DB25_Display".dbx21_1 := FALSE; END_IF;
END_REGION

REGION Network 41: Grey bar data 1: Data loaded for grey bar
   RUNG wire#powerrail
      Contact( "M91.2" )
      { S7_Templates := "SrcType := Int" } EQ_Contact(in1 := "DB03_Machine".dbw20, in2 := "DB03_Machine".dbw24)
      P_Trig( "DB01_Osr".osr61 )
      S_Coil( "DB25_Display".dbx21_1 )
   END_RUNG
   // the same network as SCL:
   #_w1 := "M91.2" AND ("DB03_Machine".dbw20 = "DB03_Machine".dbw24);
   #_w2 := #_w1 AND NOT "DB01_Osr".osr61;   // rising edge
   "DB01_Osr".osr61 := #_w1;
   IF #_w2 THEN "DB25_Display".dbx21_1 := TRUE; END_IF;
END_REGION

REGION Network 42: Rope at end of cycle selection out of range
   RUNG wire#powerrail
      { S7_GenerateENO := "TRUE" } Move(in := "DB251_ProgramDisplay".Display.RopeEndCycle, out1 => #TempInt)
   END_RUNG
   RUNG wire#powerrail
      { S7_Templates := "SrcType := Int" } GT_Contact(in1 := #TempInt, in2 := 2)
      { S7_GenerateENO := "TRUE" } Move(in := 1, out1 => "DB251_ProgramDisplay".Display.RopeEndCycle)
   END_RUNG
   // the same network as SCL:
   #TempInt := "DB251_ProgramDisplay".Display.RopeEndCycle;
   IF #TempInt > 2 THEN "DB251_ProgramDisplay".Display.RopeEndCycle := 1; END_IF;
END_REGION

REGION Network 44: Top selection out of field
   RUNG wire#powerrail
      { S7_Templates := "SrcType := Int" } LT_Contact(in1 := "DB251_ProgramDisplay".Display.Top, in2 := 1)
      wire#w1
      { S7_GenerateENO := "TRUE" } Move(in := 1, out1 => "DB251_ProgramDisplay".Display.Top)
   END_RUNG
   RUNG wire#powerrail
      { S7_Templates := "SrcType := Int" } GT_Contact(in1 := "DB251_ProgramDisplay".Display.Top, in2 := 9)
   END_RUNG wire#w1
   // the same network as SCL:
   IF ("DB251_ProgramDisplay".Display.Top < 1) OR ("DB251_ProgramDisplay".Display.Top > 9) THEN
       "DB251_ProgramDisplay".Display.Top := 1;
   END_IF;
END_REGION

REGION Network 45: Top film lenght out of range
   RUNG wire#powerrail
      { S7_Templates := "SrcType := Int" } LE_Contact(in1 := "DB251_ProgramDisplay".Display.TopLenght, in2 := 500)
      { S7_GenerateENO := "TRUE" } Move(in := 500, out1 => "DB251_ProgramDisplay".Display.TopLenght)
   END_RUNG
   // the same network as SCL:
   IF "DB251_ProgramDisplay".Display.TopLenght <= 500 THEN
       "DB251_ProgramDisplay".Display.TopLenght := 500;
   END_IF;
END_REGION

REGION Network 46: Band unit out of range (1-6)
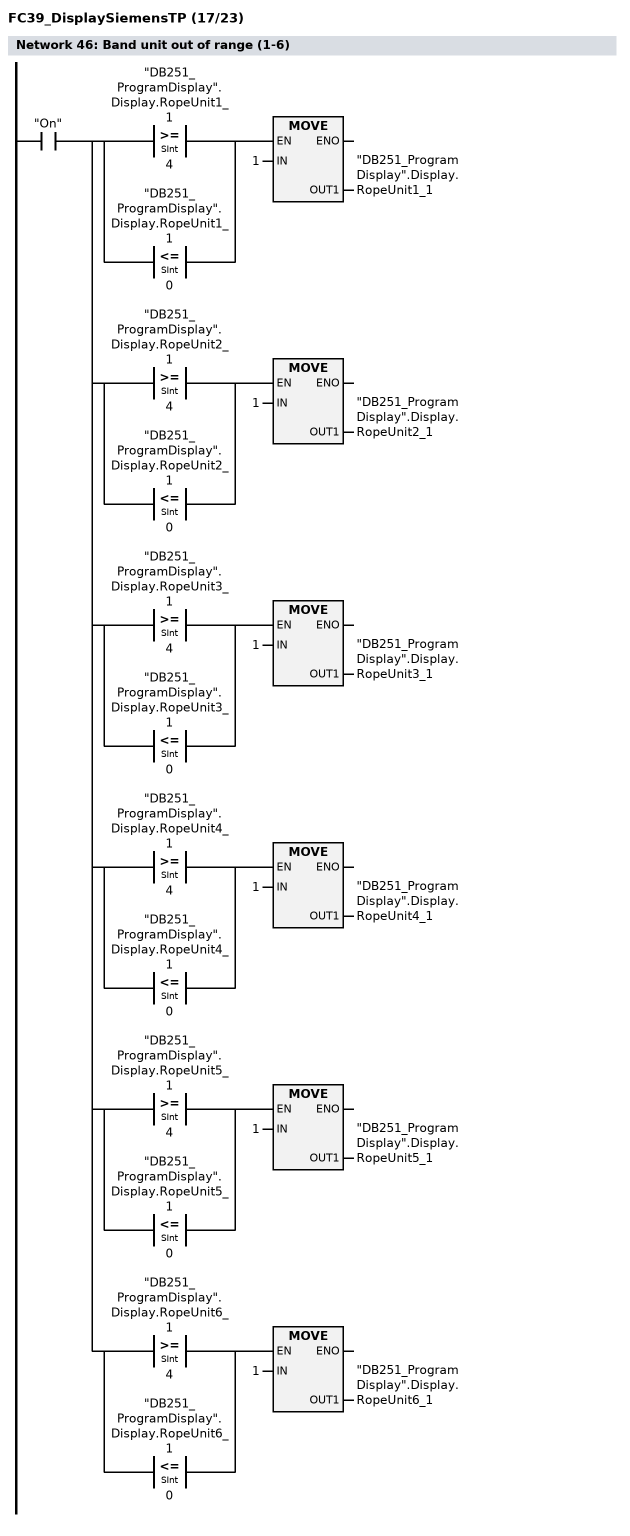
   RUNG wire#powerrail
      Contact( "On" )
      wire#w1
      { S7_Templates := "SrcType := SInt" } GE_Contact(in1 := "DB251_ProgramDisplay".Display.RopeUnit1_1, in2 := 4)
      wire#w2
      { S7_GenerateENO := "TRUE" } Move(in := 1, out1 => "DB251_ProgramDisplay".Display.RopeUnit1_1)
   END_RUNG
   RUNG wire#w1
      { S7_Templates := "SrcType := SInt" } LE_Contact(in1 := "DB251_ProgramDisplay".Display.RopeUnit1_1, in2 := 0)
   END_RUNG wire#w2
   RUNG wire#w1
      { S7_Templates := "SrcType := SInt" } GE_Contact(in1 := "DB251_ProgramDisplay".Display.RopeUnit2_1, in2 := 4)
      wire#w3
      { S7_GenerateENO := "TRUE" } Move(in := 1, out1 => "DB251_ProgramDisplay".Display.RopeUnit2_1)
   END_RUNG
   RUNG wire#w1
      { S7_Templates := "SrcType := SInt" } LE_Contact(in1 := "DB251_ProgramDisplay".Display.RopeUnit2_1, in2 := 0)
   END_RUNG wire#w3
   RUNG wire#w1
      { S7_Templates := "SrcType := SInt" } GE_Contact(in1 := "DB251_ProgramDisplay".Display.RopeUnit3_1, in2 := 4)
      wire#w4
      { S7_GenerateENO := "TRUE" } Move(in := 1, out1 => "DB251_ProgramDisplay".Display.RopeUnit3_1)
   END_RUNG
   RUNG wire#w1
      { S7_Templates := "SrcType := SInt" } LE_Contact(in1 := "DB251_ProgramDisplay".Display.RopeUnit3_1, in2 := 0)
   END_RUNG wire#w4
   RUNG wire#w1
      { S7_Templates := "SrcType := SInt" } GE_Contact(in1 := "DB251_ProgramDisplay".Display.RopeUnit4_1, in2 := 4)
      wire#w5
      { S7_GenerateENO := "TRUE" } Move(in := 1, out1 => "DB251_ProgramDisplay".Display.RopeUnit4_1)
   END_RUNG
   RUNG wire#w1
      { S7_Templates := "SrcType := SInt" } LE_Contact(in1 := "DB251_ProgramDisplay".Display.RopeUnit4_1, in2 := 0)
   END_RUNG wire#w5
   RUNG wire#w1
      { S7_Templates := "SrcType := SInt" } GE_Contact(in1 := "DB251_ProgramDisplay".Display.RopeUnit5_1, in2 := 4)
      wire#w6
      { S7_GenerateENO := "TRUE" } Move(in := 1, out1 => "DB251_ProgramDisplay".Display.RopeUnit5_1)
   END_RUNG
   RUNG wire#w1
      { S7_Templates := "SrcType := SInt" } LE_Contact(in1 := "DB251_ProgramDisplay".Display.RopeUnit5_1, in2 := 0)
   END_RUNG wire#w6
   RUNG wire#w1
      { S7_Templates := "SrcType := SInt" } GE_Contact(in1 := "DB251_ProgramDisplay".Display.RopeUnit6_1, in2 := 4)
      wire#w7
      { S7_GenerateENO := "TRUE" } Move(in := 1, out1 => "DB251_ProgramDisplay".Display.RopeUnit6_1)
   END_RUNG
   RUNG wire#w1
      { S7_Templates := "SrcType := SInt" } LE_Contact(in1 := "DB251_ProgramDisplay".Display.RopeUnit6_1, in2 := 0)
   END_RUNG wire#w7
   // the same network as SCL:
   IF "On" AND (("DB251_ProgramDisplay".Display.RopeUnit1_1 >= 4) OR ("DB251_ProgramDisplay".Display.RopeUnit1_1 <= 0)) THEN
       "DB251_ProgramDisplay".Display.RopeUnit1_1 := 1;
   END_IF;
   IF "On" AND (("DB251_ProgramDisplay".Display.RopeUnit2_1 >= 4) OR ("DB251_ProgramDisplay".Display.RopeUnit2_1 <= 0)) THEN
       "DB251_ProgramDisplay".Display.RopeUnit2_1 := 1;
   END_IF;
   IF "On" AND (("DB251_ProgramDisplay".Display.RopeUnit3_1 >= 4) OR ("DB251_ProgramDisplay".Display.RopeUnit3_1 <= 0)) THEN
       "DB251_ProgramDisplay".Display.RopeUnit3_1 := 1;
   END_IF;
   IF "On" AND (("DB251_ProgramDisplay".Display.RopeUnit4_1 >= 4) OR ("DB251_ProgramDisplay".Display.RopeUnit4_1 <= 0)) THEN
       "DB251_ProgramDisplay".Display.RopeUnit4_1 := 1;
   END_IF;
   IF "On" AND (("DB251_ProgramDisplay".Display.RopeUnit5_1 >= 4) OR ("DB251_ProgramDisplay".Display.RopeUnit5_1 <= 0)) THEN
       "DB251_ProgramDisplay".Display.RopeUnit5_1 := 1;
   END_IF;
   IF "On" AND (("DB251_ProgramDisplay".Display.RopeUnit6_1 >= 4) OR ("DB251_ProgramDisplay".Display.RopeUnit6_1 <= 0)) THEN
       "DB251_ProgramDisplay".Display.RopeUnit6_1 := 1;
   END_IF;
END_REGION

REGION Network 47: Band unit out of range (7-12)
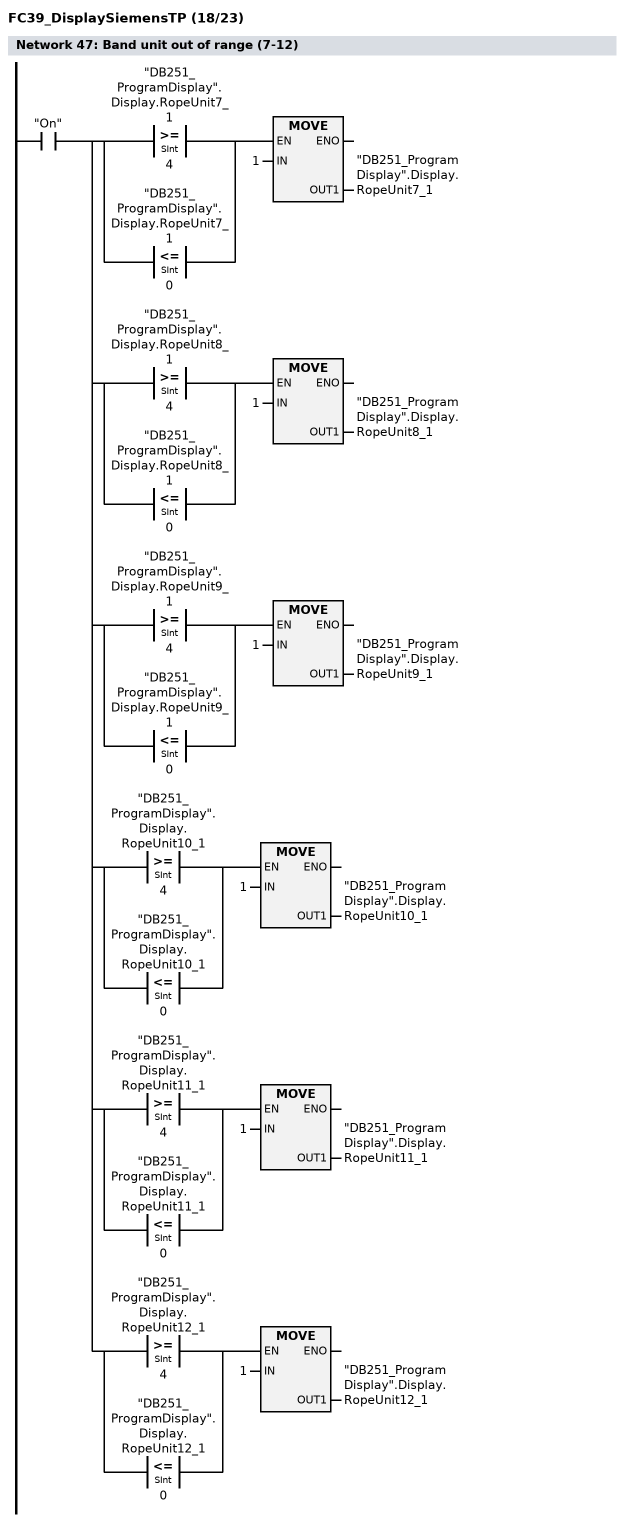
   RUNG wire#powerrail
      Contact( "On" )
      wire#w1
      { S7_Templates := "SrcType := SInt" } GE_Contact(in1 := "DB251_ProgramDisplay".Display.RopeUnit7_1, in2 := 4)
      wire#w2
      { S7_GenerateENO := "TRUE" } Move(in := 1, out1 => "DB251_ProgramDisplay".Display.RopeUnit7_1)
   END_RUNG
   RUNG wire#w1
      { S7_Templates := "SrcType := SInt" } LE_Contact(in1 := "DB251_ProgramDisplay".Display.RopeUnit7_1, in2 := 0)
   END_RUNG wire#w2
   RUNG wire#w1
      { S7_Templates := "SrcType := SInt" } GE_Contact(in1 := "DB251_ProgramDisplay".Display.RopeUnit8_1, in2 := 4)
      wire#w3
      { S7_GenerateENO := "TRUE" } Move(in := 1, out1 => "DB251_ProgramDisplay".Display.RopeUnit8_1)
   END_RUNG
   RUNG wire#w1
      { S7_Templates := "SrcType := SInt" } LE_Contact(in1 := "DB251_ProgramDisplay".Display.RopeUnit8_1, in2 := 0)
   END_RUNG wire#w3
   RUNG wire#w1
      { S7_Templates := "SrcType := SInt" } GE_Contact(in1 := "DB251_ProgramDisplay".Display.RopeUnit9_1, in2 := 4)
      wire#w4
      { S7_GenerateENO := "TRUE" } Move(in := 1, out1 => "DB251_ProgramDisplay".Display.RopeUnit9_1)
   END_RUNG
   RUNG wire#w1
      { S7_Templates := "SrcType := SInt" } LE_Contact(in1 := "DB251_ProgramDisplay".Display.RopeUnit9_1, in2 := 0)
   END_RUNG wire#w4
   RUNG wire#w1
      { S7_Templates := "SrcType := SInt" } GE_Contact(in1 := "DB251_ProgramDisplay".Display.RopeUnit10_1, in2 := 4)
      wire#w5
      { S7_GenerateENO := "TRUE" } Move(in := 1, out1 => "DB251_ProgramDisplay".Display.RopeUnit10_1)
   END_RUNG
   RUNG wire#w1
      { S7_Templates := "SrcType := SInt" } LE_Contact(in1 := "DB251_ProgramDisplay".Display.RopeUnit10_1, in2 := 0)
   END_RUNG wire#w5
   RUNG wire#w1
      { S7_Templates := "SrcType := SInt" } GE_Contact(in1 := "DB251_ProgramDisplay".Display.RopeUnit11_1, in2 := 4)
      wire#w6
      { S7_GenerateENO := "TRUE" } Move(in := 1, out1 => "DB251_ProgramDisplay".Display.RopeUnit11_1)
   END_RUNG
   RUNG wire#w1
      { S7_Templates := "SrcType := SInt" } LE_Contact(in1 := "DB251_ProgramDisplay".Display.RopeUnit11_1, in2 := 0)
   END_RUNG wire#w6
   RUNG wire#w1
      { S7_Templates := "SrcType := SInt" } GE_Contact(in1 := "DB251_ProgramDisplay".Display.RopeUnit12_1, in2 := 4)
      wire#w7
      { S7_GenerateENO := "TRUE" } Move(in := 1, out1 => "DB251_ProgramDisplay".Display.RopeUnit12_1)
   END_RUNG
   RUNG wire#w1
      { S7_Templates := "SrcType := SInt" } LE_Contact(in1 := "DB251_ProgramDisplay".Display.RopeUnit12_1, in2 := 0)
   END_RUNG wire#w7
   // the same network as SCL:
   IF "On" AND (("DB251_ProgramDisplay".Display.RopeUnit7_1 >= 4) OR ("DB251_ProgramDisplay".Display.RopeUnit7_1 <= 0)) THEN
       "DB251_ProgramDisplay".Display.RopeUnit7_1 := 1;
   END_IF;
   IF "On" AND (("DB251_ProgramDisplay".Display.RopeUnit8_1 >= 4) OR ("DB251_ProgramDisplay".Display.RopeUnit8_1 <= 0)) THEN
       "DB251_ProgramDisplay".Display.RopeUnit8_1 := 1;
   END_IF;
   IF "On" AND (("DB251_ProgramDisplay".Display.RopeUnit9_1 >= 4) OR ("DB251_ProgramDisplay".Display.RopeUnit9_1 <= 0)) THEN
       "DB251_ProgramDisplay".Display.RopeUnit9_1 := 1;
   END_IF;
   IF "On" AND (("DB251_ProgramDisplay".Display.RopeUnit10_1 >= 4) OR ("DB251_ProgramDisplay".Display.RopeUnit10_1 <= 0)) THEN
       "DB251_ProgramDisplay".Display.RopeUnit10_1 := 1;
   END_IF;
   IF "On" AND (("DB251_ProgramDisplay".Display.RopeUnit11_1 >= 4) OR ("DB251_ProgramDisplay".Display.RopeUnit11_1 <= 0)) THEN
       "DB251_ProgramDisplay".Display.RopeUnit11_1 := 1;
   END_IF;
   IF "On" AND (("DB251_ProgramDisplay".Display.RopeUnit12_1 >= 4) OR ("DB251_ProgramDisplay".Display.RopeUnit12_1 <= 0)) THEN
       "DB251_ProgramDisplay".Display.RopeUnit12_1 := 1;
   END_IF;
END_REGION

REGION Network 48: Rope unit out of range (1-6)
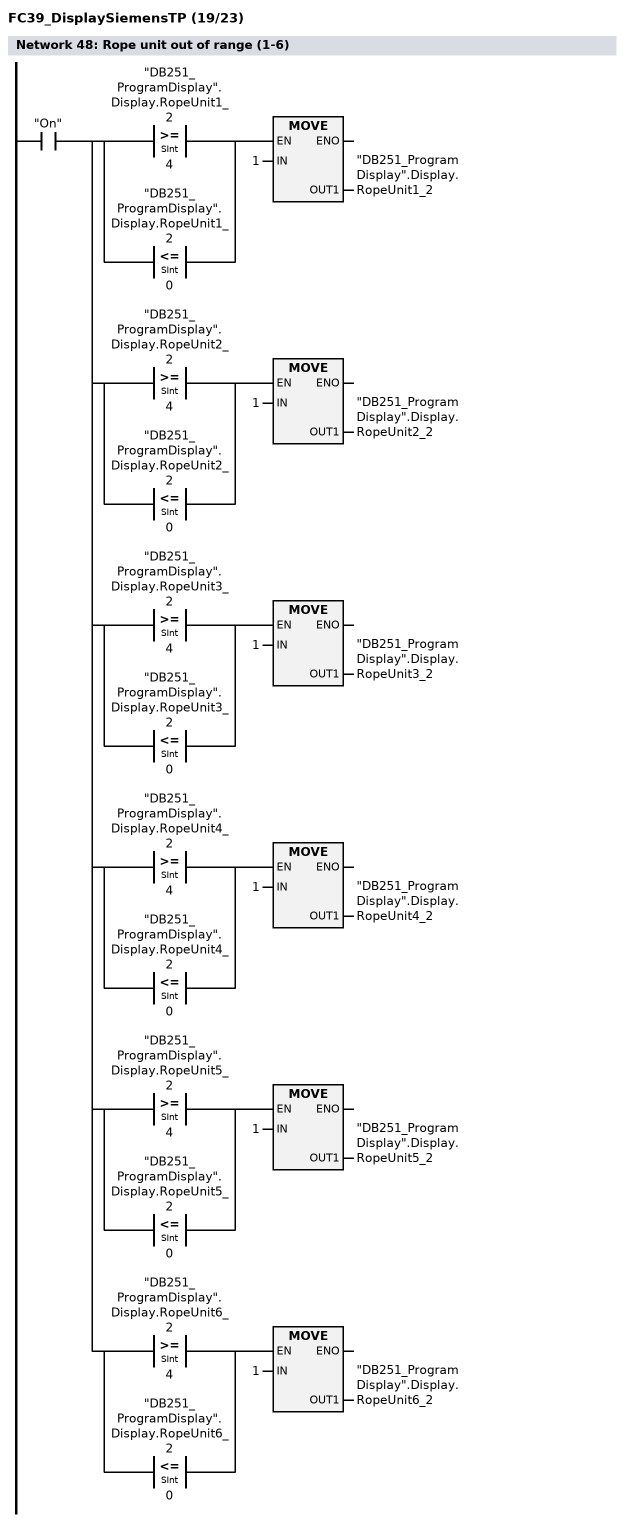
   RUNG wire#powerrail
      Contact( "On" )
      wire#w1
      { S7_Templates := "SrcType := SInt" } GE_Contact(in1 := "DB251_ProgramDisplay".Display.RopeUnit1_2, in2 := 4)
      wire#w2
      { S7_GenerateENO := "TRUE" } Move(in := 1, out1 => "DB251_ProgramDisplay".Display.RopeUnit1_2)
   END_RUNG
   RUNG wire#w1
      { S7_Templates := "SrcType := SInt" } LE_Contact(in1 := "DB251_ProgramDisplay".Display.RopeUnit1_2, in2 := 0)
   END_RUNG wire#w2
   RUNG wire#w1
      { S7_Templates := "SrcType := SInt" } GE_Contact(in1 := "DB251_ProgramDisplay".Display.RopeUnit2_2, in2 := 4)
      wire#w3
      { S7_GenerateENO := "TRUE" } Move(in := 1, out1 => "DB251_ProgramDisplay".Display.RopeUnit2_2)
   END_RUNG
   RUNG wire#w1
      { S7_Templates := "SrcType := SInt" } LE_Contact(in1 := "DB251_ProgramDisplay".Display.RopeUnit2_2, in2 := 0)
   END_RUNG wire#w3
   RUNG wire#w1
      { S7_Templates := "SrcType := SInt" } GE_Contact(in1 := "DB251_ProgramDisplay".Display.RopeUnit3_2, in2 := 4)
      wire#w4
      { S7_GenerateENO := "TRUE" } Move(in := 1, out1 => "DB251_ProgramDisplay".Display.RopeUnit3_2)
   END_RUNG
   RUNG wire#w1
      { S7_Templates := "SrcType := SInt" } LE_Contact(in1 := "DB251_ProgramDisplay".Display.RopeUnit3_2, in2 := 0)
   END_RUNG wire#w4
   RUNG wire#w1
      { S7_Templates := "SrcType := SInt" } GE_Contact(in1 := "DB251_ProgramDisplay".Display.RopeUnit4_2, in2 := 4)
      wire#w5
      { S7_GenerateENO := "TRUE" } Move(in := 1, out1 => "DB251_ProgramDisplay".Display.RopeUnit4_2)
   END_RUNG
   RUNG wire#w1
      { S7_Templates := "SrcType := SInt" } LE_Contact(in1 := "DB251_ProgramDisplay".Display.RopeUnit4_2, in2 := 0)
   END_RUNG wire#w5
   RUNG wire#w1
      { S7_Templates := "SrcType := SInt" } GE_Contact(in1 := "DB251_ProgramDisplay".Display.RopeUnit5_2, in2 := 4)
      wire#w6
      { S7_GenerateENO := "TRUE" } Move(in := 1, out1 => "DB251_ProgramDisplay".Display.RopeUnit5_2)
   END_RUNG
   RUNG wire#w1
      { S7_Templates := "SrcType := SInt" } LE_Contact(in1 := "DB251_ProgramDisplay".Display.RopeUnit5_2, in2 := 0)
   END_RUNG wire#w6
   RUNG wire#w1
      { S7_Templates := "SrcType := SInt" } GE_Contact(in1 := "DB251_ProgramDisplay".Display.RopeUnit6_2, in2 := 4)
      wire#w7
      { S7_GenerateENO := "TRUE" } Move(in := 1, out1 => "DB251_ProgramDisplay".Display.RopeUnit6_2)
   END_RUNG
   RUNG wire#w1
      { S7_Templates := "SrcType := SInt" } LE_Contact(in1 := "DB251_ProgramDisplay".Display.RopeUnit6_2, in2 := 0)
   END_RUNG wire#w7
   // the same network as SCL:
   IF "On" AND (("DB251_ProgramDisplay".Display.RopeUnit1_2 >= 4) OR ("DB251_ProgramDisplay".Display.RopeUnit1_2 <= 0)) THEN
       "DB251_ProgramDisplay".Display.RopeUnit1_2 := 1;
   END_IF;
   IF "On" AND (("DB251_ProgramDisplay".Display.RopeUnit2_2 >= 4) OR ("DB251_ProgramDisplay".Display.RopeUnit2_2 <= 0)) THEN
       "DB251_ProgramDisplay".Display.RopeUnit2_2 := 1;
   END_IF;
   IF "On" AND (("DB251_ProgramDisplay".Display.RopeUnit3_2 >= 4) OR ("DB251_ProgramDisplay".Display.RopeUnit3_2 <= 0)) THEN
       "DB251_ProgramDisplay".Display.RopeUnit3_2 := 1;
   END_IF;
   IF "On" AND (("DB251_ProgramDisplay".Display.RopeUnit4_2 >= 4) OR ("DB251_ProgramDisplay".Display.RopeUnit4_2 <= 0)) THEN
       "DB251_ProgramDisplay".Display.RopeUnit4_2 := 1;
   END_IF;
   IF "On" AND (("DB251_ProgramDisplay".Display.RopeUnit5_2 >= 4) OR ("DB251_ProgramDisplay".Display.RopeUnit5_2 <= 0)) THEN
       "DB251_ProgramDisplay".Display.RopeUnit5_2 := 1;
   END_IF;
   IF "On" AND (("DB251_ProgramDisplay".Display.RopeUnit6_2 >= 4) OR ("DB251_ProgramDisplay".Display.RopeUnit6_2 <= 0)) THEN
       "DB251_ProgramDisplay".Display.RopeUnit6_2 := 1;
   END_IF;
END_REGION

REGION Network 49: Rope unit out of range (7-12)
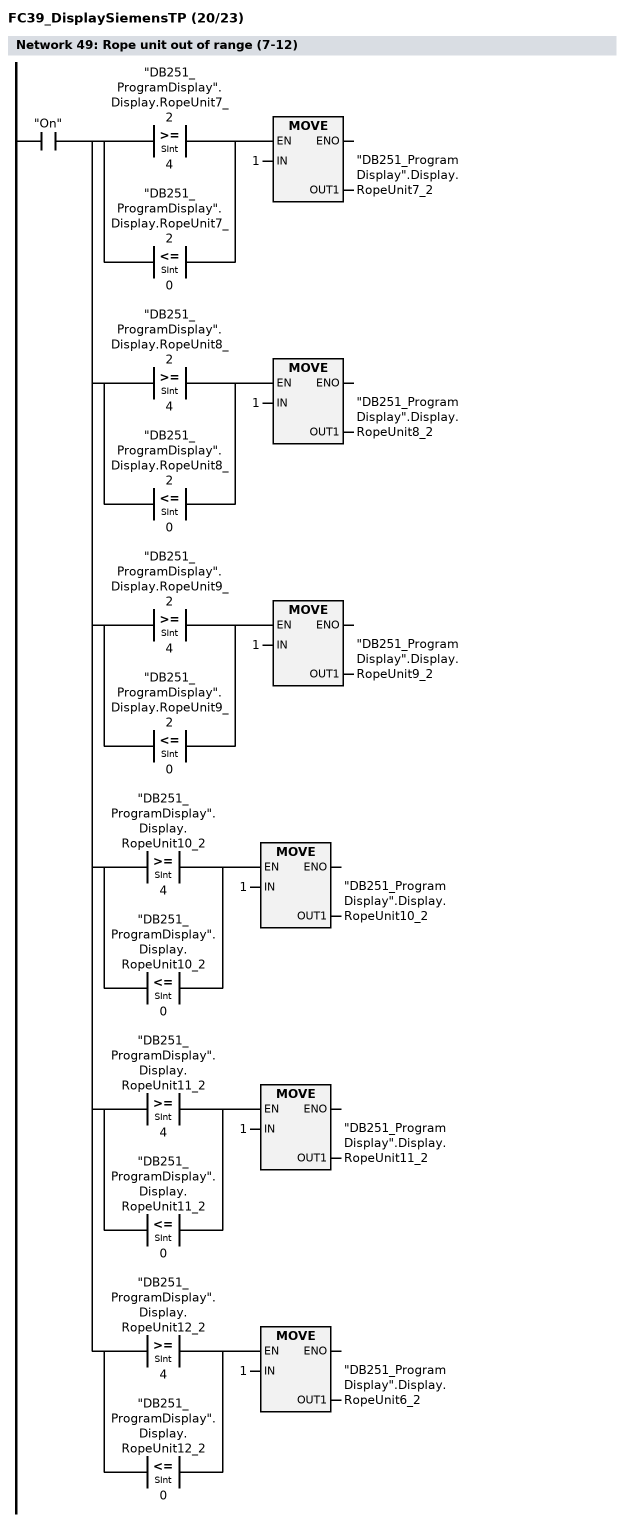
   RUNG wire#powerrail
      Contact( "On" )
      wire#w1
      { S7_Templates := "SrcType := SInt" } GE_Contact(in1 := "DB251_ProgramDisplay".Display.RopeUnit7_2, in2 := 4)
      wire#w2
      { S7_GenerateENO := "TRUE" } Move(in := 1, out1 => "DB251_ProgramDisplay".Display.RopeUnit7_2)
   END_RUNG
   RUNG wire#w1
      { S7_Templates := "SrcType := SInt" } LE_Contact(in1 := "DB251_ProgramDisplay".Display.RopeUnit7_2, in2 := 0)
   END_RUNG wire#w2
   RUNG wire#w1
      { S7_Templates := "SrcType := SInt" } GE_Contact(in1 := "DB251_ProgramDisplay".Display.RopeUnit8_2, in2 := 4)
      wire#w3
      { S7_GenerateENO := "TRUE" } Move(in := 1, out1 => "DB251_ProgramDisplay".Display.RopeUnit8_2)
   END_RUNG
   RUNG wire#w1
      { S7_Templates := "SrcType := SInt" } LE_Contact(in1 := "DB251_ProgramDisplay".Display.RopeUnit8_2, in2 := 0)
   END_RUNG wire#w3
   RUNG wire#w1
      { S7_Templates := "SrcType := SInt" } GE_Contact(in1 := "DB251_ProgramDisplay".Display.RopeUnit9_2, in2 := 4)
      wire#w4
      { S7_GenerateENO := "TRUE" } Move(in := 1, out1 => "DB251_ProgramDisplay".Display.RopeUnit9_2)
   END_RUNG
   RUNG wire#w1
      { S7_Templates := "SrcType := SInt" } LE_Contact(in1 := "DB251_ProgramDisplay".Display.RopeUnit9_2, in2 := 0)
   END_RUNG wire#w4
   RUNG wire#w1
      { S7_Templates := "SrcType := SInt" } GE_Contact(in1 := "DB251_ProgramDisplay".Display.RopeUnit10_2, in2 := 4)
      wire#w5
      { S7_GenerateENO := "TRUE" } Move(in := 1, out1 => "DB251_ProgramDisplay".Display.RopeUnit10_2)
   END_RUNG
   RUNG wire#w1
      { S7_Templates := "SrcType := SInt" } LE_Contact(in1 := "DB251_ProgramDisplay".Display.RopeUnit10_2, in2 := 0)
   END_RUNG wire#w5
   RUNG wire#w1
      { S7_Templates := "SrcType := SInt" } GE_Contact(in1 := "DB251_ProgramDisplay".Display.RopeUnit11_2, in2 := 4)
      wire#w6
      { S7_GenerateENO := "TRUE" } Move(in := 1, out1 => "DB251_ProgramDisplay".Display.RopeUnit11_2)
   END_RUNG
   RUNG wire#w1
      { S7_Templates := "SrcType := SInt" } LE_Contact(in1 := "DB251_ProgramDisplay".Display.RopeUnit11_2, in2 := 0)
   END_RUNG wire#w6
   RUNG wire#w1
      { S7_Templates := "SrcType := SInt" } GE_Contact(in1 := "DB251_ProgramDisplay".Display.RopeUnit12_2, in2 := 4)
      wire#w7
      { S7_GenerateENO := "TRUE" } Move(in := 1, out1 => "DB251_ProgramDisplay".Display.RopeUnit6_2)
   END_RUNG
   RUNG wire#w1
      { S7_Templates := "SrcType := SInt" } LE_Contact(in1 := "DB251_ProgramDisplay".Display.RopeUnit12_2, in2 := 0)
   END_RUNG wire#w7
   // the same network as SCL:
   IF "On" AND (("DB251_ProgramDisplay".Display.RopeUnit7_2 >= 4) OR ("DB251_ProgramDisplay".Display.RopeUnit7_2 <= 0)) THEN
       "DB251_ProgramDisplay".Display.RopeUnit7_2 := 1;
   END_IF;
   IF "On" AND (("DB251_ProgramDisplay".Display.RopeUnit8_2 >= 4) OR ("DB251_ProgramDisplay".Display.RopeUnit8_2 <= 0)) THEN
       "DB251_ProgramDisplay".Display.RopeUnit8_2 := 1;
   END_IF;
   IF "On" AND (("DB251_ProgramDisplay".Display.RopeUnit9_2 >= 4) OR ("DB251_ProgramDisplay".Display.RopeUnit9_2 <= 0)) THEN
       "DB251_ProgramDisplay".Display.RopeUnit9_2 := 1;
   END_IF;
   IF "On" AND (("DB251_ProgramDisplay".Display.RopeUnit10_2 >= 4) OR ("DB251_ProgramDisplay".Display.RopeUnit10_2 <= 0)) THEN
       "DB251_ProgramDisplay".Display.RopeUnit10_2 := 1;
   END_IF;
   IF "On" AND (("DB251_ProgramDisplay".Display.RopeUnit11_2 >= 4) OR ("DB251_ProgramDisplay".Display.RopeUnit11_2 <= 0)) THEN
       "DB251_ProgramDisplay".Display.RopeUnit11_2 := 1;
   END_IF;
   IF "On" AND (("DB251_ProgramDisplay".Display.RopeUnit12_2 >= 4) OR ("DB251_ProgramDisplay".Display.RopeUnit12_2 <= 0)) THEN
       "DB251_ProgramDisplay".Display.RopeUnit6_2 := 1;
   END_IF;
END_REGION

REGION Network 50: Define landmark to bottom for the last step
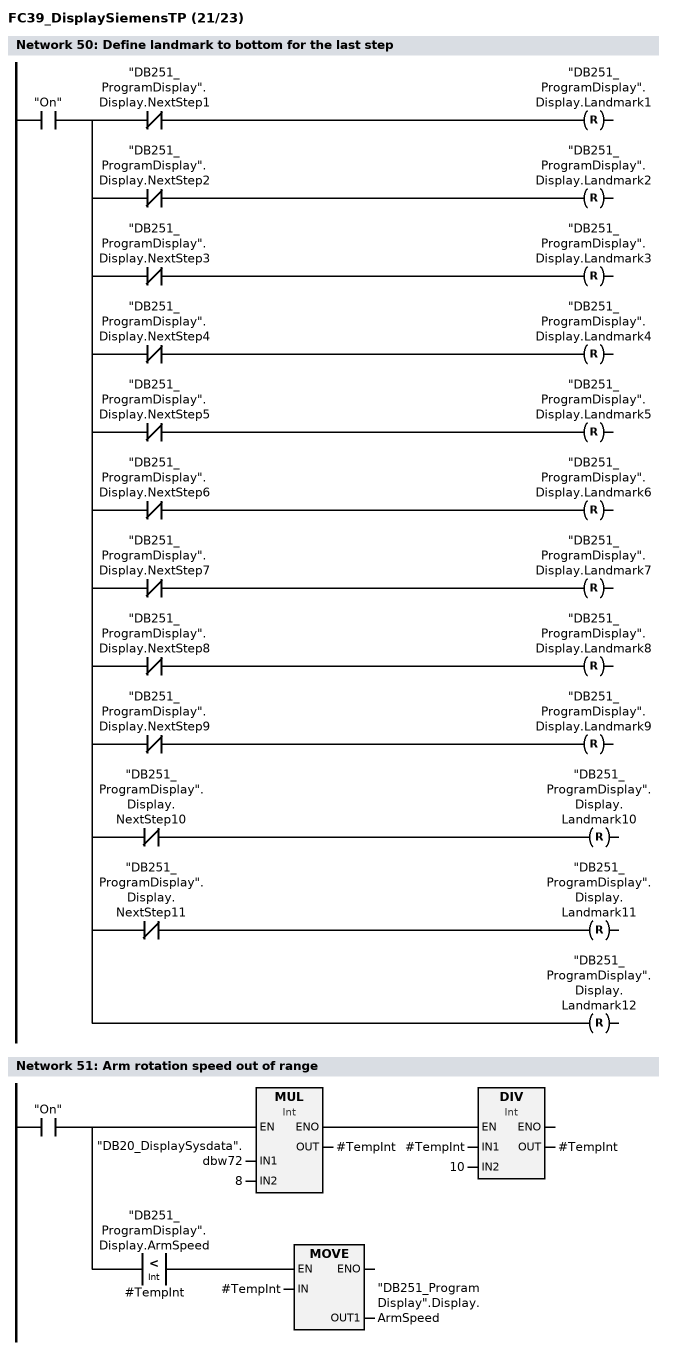
   RUNG wire#powerrail
      Contact( "On" )
      wire#w1
      I_Contact( "DB251_ProgramDisplay".Display.NextStep1 )
      R_Coil( "DB251_ProgramDisplay".Display.Landmark1 )
   END_RUNG
   RUNG wire#w1
      I_Contact( "DB251_ProgramDisplay".Display.NextStep2 )
      R_Coil( "DB251_ProgramDisplay".Display.Landmark2 )
   END_RUNG
   RUNG wire#w1
      I_Contact( "DB251_ProgramDisplay".Display.NextStep3 )
      R_Coil( "DB251_ProgramDisplay".Display.Landmark3 )
   END_RUNG
   RUNG wire#w1
      I_Contact( "DB251_ProgramDisplay".Display.NextStep4 )
      R_Coil( "DB251_ProgramDisplay".Display.Landmark4 )
   END_RUNG
   RUNG wire#w1
      I_Contact( "DB251_ProgramDisplay".Display.NextStep5 )
      R_Coil( "DB251_ProgramDisplay".Display.Landmark5 )
   END_RUNG
   RUNG wire#w1
      I_Contact( "DB251_ProgramDisplay".Display.NextStep6 )
      R_Coil( "DB251_ProgramDisplay".Display.Landmark6 )
   END_RUNG
   RUNG wire#w1
      I_Contact( "DB251_ProgramDisplay".Display.NextStep7 )
      R_Coil( "DB251_ProgramDisplay".Display.Landmark7 )
   END_RUNG
   RUNG wire#w1
      I_Contact( "DB251_ProgramDisplay".Display.NextStep8 )
      R_Coil( "DB251_ProgramDisplay".Display.Landmark8 )
   END_RUNG
   RUNG wire#w1
      I_Contact( "DB251_ProgramDisplay".Display.NextStep9 )
      R_Coil( "DB251_ProgramDisplay".Display.Landmark9 )
   END_RUNG
   RUNG wire#w1
      I_Contact( "DB251_ProgramDisplay".Display.NextStep10 )
      R_Coil( "DB251_ProgramDisplay".Display.Landmark10 )
   END_RUNG
   RUNG wire#w1
      I_Contact( "DB251_ProgramDisplay".Display.NextStep11 )
      R_Coil( "DB251_ProgramDisplay".Display.Landmark11 )
   END_RUNG
   RUNG wire#w1
      R_Coil( "DB251_ProgramDisplay".Display.Landmark12 )
   END_RUNG
   // the same network as SCL:
   IF "On" AND NOT "DB251_ProgramDisplay".Display.NextStep1 THEN
       "DB251_ProgramDisplay".Display.Landmark1 := FALSE;
   END_IF;
   IF "On" AND NOT "DB251_ProgramDisplay".Display.NextStep2 THEN
       "DB251_ProgramDisplay".Display.Landmark2 := FALSE;
   END_IF;
   IF "On" AND NOT "DB251_ProgramDisplay".Display.NextStep3 THEN
       "DB251_ProgramDisplay".Display.Landmark3 := FALSE;
   END_IF;
   IF "On" AND NOT "DB251_ProgramDisplay".Display.NextStep4 THEN
       "DB251_ProgramDisplay".Display.Landmark4 := FALSE;
   END_IF;
   IF "On" AND NOT "DB251_ProgramDisplay".Display.NextStep5 THEN
       "DB251_ProgramDisplay".Display.Landmark5 := FALSE;
   END_IF;
   IF "On" AND NOT "DB251_ProgramDisplay".Display.NextStep6 THEN
       "DB251_ProgramDisplay".Display.Landmark6 := FALSE;
   END_IF;
   IF "On" AND NOT "DB251_ProgramDisplay".Display.NextStep7 THEN
       "DB251_ProgramDisplay".Display.Landmark7 := FALSE;
   END_IF;
   IF "On" AND NOT "DB251_ProgramDisplay".Display.NextStep8 THEN
       "DB251_ProgramDisplay".Display.Landmark8 := FALSE;
   END_IF;
   IF "On" AND NOT "DB251_ProgramDisplay".Display.NextStep9 THEN
       "DB251_ProgramDisplay".Display.Landmark9 := FALSE;
   END_IF;
   IF "On" AND NOT "DB251_ProgramDisplay".Display.NextStep10 THEN
       "DB251_ProgramDisplay".Display.Landmark10 := FALSE;
   END_IF;
   IF "On" AND NOT "DB251_ProgramDisplay".Display.NextStep11 THEN
       "DB251_ProgramDisplay".Display.Landmark11 := FALSE;
   END_IF;
   IF "On" THEN "DB251_ProgramDisplay".Display.Landmark12 := FALSE; END_IF;
END_REGION

REGION Network 51: Arm rotation speed out of range
   RUNG wire#powerrail
      Contact( "On" )
      wire#w1
      { S7_Templates := "SrcType := Int"; S7_GenerateENO := "TRUE" } Mul(in1 := "DB20_DisplaySysdata".dbw72, in2 := 8, out => #TempInt)
      { S7_Templates := "SrcType := Int"; S7_GenerateENO := "TRUE" } Div(in1 := #TempInt, in2 := 10, out => #TempInt)
   END_RUNG
   RUNG wire#w1
      { S7_Templates := "SrcType := Int" } LT_Contact(in1 := "DB251_ProgramDisplay".Display.ArmSpeed, in2 := #TempInt)
      { S7_GenerateENO := "TRUE" } Move(in := #TempInt, out1 => "DB251_ProgramDisplay".Display.ArmSpeed)
   END_RUNG
   // the same network as SCL:
   // ENO of a box is taken as its EN; it also drops when the box reports an error
   IF "On" THEN
       #TempInt := "DB20_DisplaySysdata".dbw72 * 8;
       #TempInt := #TempInt / 10;
   END_IF;
   IF "On" AND ("DB251_ProgramDisplay".Display.ArmSpeed < #TempInt) THEN
       "DB251_ProgramDisplay".Display.ArmSpeed := #TempInt;
   END_IF;
END_REGION

REGION Network 52: Next step for spool carriage height 12 (0=End 1=Next)
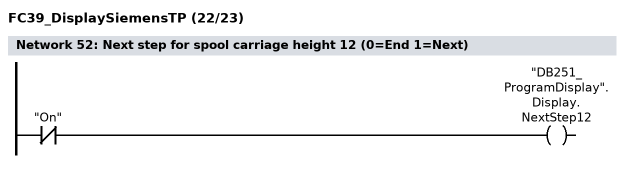
   RUNG wire#powerrail
      I_Contact( "On" )
      Coil( "DB251_ProgramDisplay".Display.NextStep12 )
   END_RUNG
   // the same network as SCL:
   "DB251_ProgramDisplay".Display.NextStep12 := NOT "On";
END_REGION

REGION Network 53
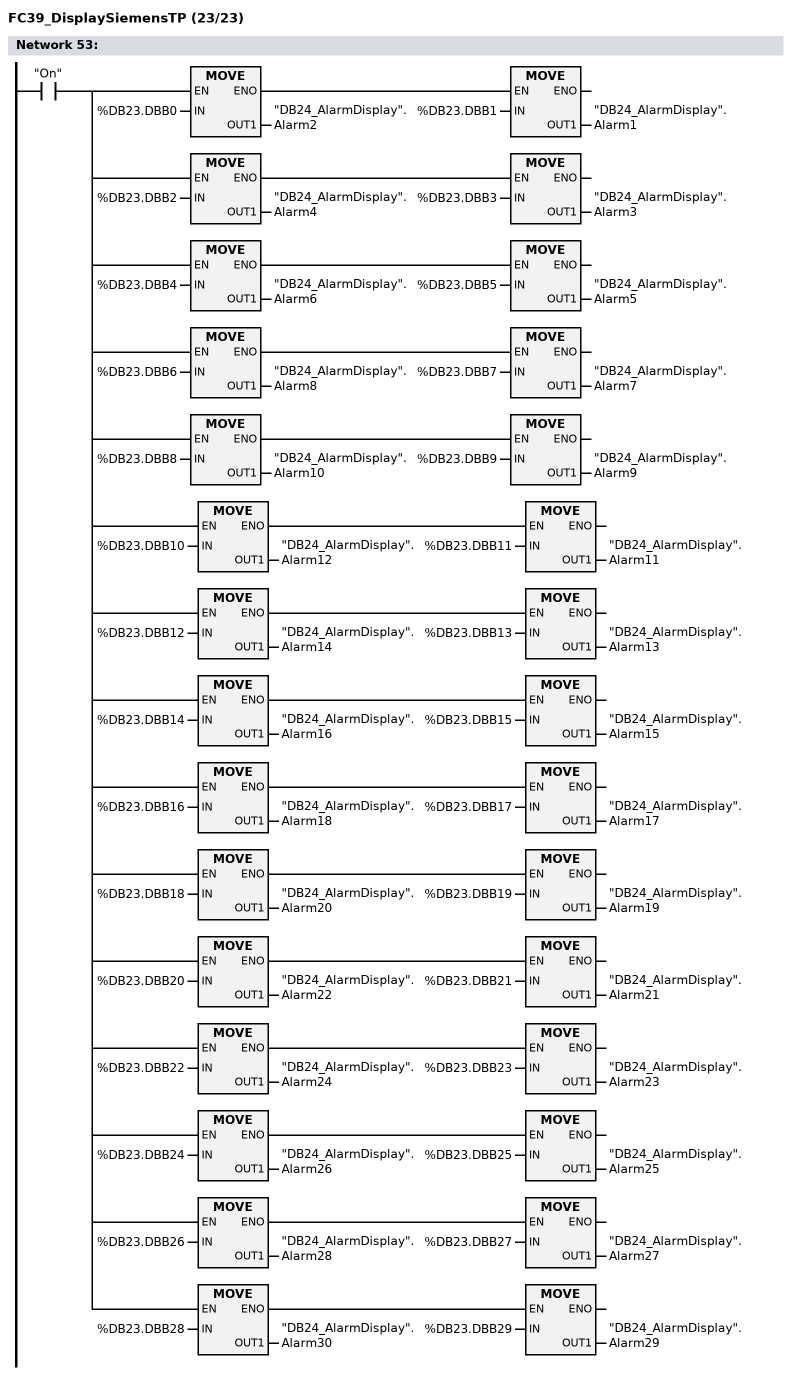
   RUNG wire#powerrail
      Contact( "On" )
      wire#w1
      { S7_GenerateENO := "TRUE" } Move(in := %DB23.DBB0, out1 => "DB24_AlarmDisplay".Alarm2)
      { S7_GenerateENO := "TRUE" } Move(in := %DB23.DBB1, out1 => "DB24_AlarmDisplay".Alarm1)
   END_RUNG
   RUNG wire#w1
      { S7_GenerateENO := "TRUE" } Move(in := %DB23.DBB2, out1 => "DB24_AlarmDisplay".Alarm4)
      { S7_GenerateENO := "TRUE" } Move(in := %DB23.DBB3, out1 => "DB24_AlarmDisplay".Alarm3)
   END_RUNG
   RUNG wire#w1
      { S7_GenerateENO := "TRUE" } Move(in := %DB23.DBB4, out1 => "DB24_AlarmDisplay".Alarm6)
      { S7_GenerateENO := "TRUE" } Move(in := %DB23.DBB5, out1 => "DB24_AlarmDisplay".Alarm5)
   END_RUNG
   RUNG wire#w1
      { S7_GenerateENO := "TRUE" } Move(in := %DB23.DBB6, out1 => "DB24_AlarmDisplay".Alarm8)
      { S7_GenerateENO := "TRUE" } Move(in := %DB23.DBB7, out1 => "DB24_AlarmDisplay".Alarm7)
   END_RUNG
   RUNG wire#w1
      { S7_GenerateENO := "TRUE" } Move(in := %DB23.DBB8, out1 => "DB24_AlarmDisplay".Alarm10)
      { S7_GenerateENO := "TRUE" } Move(in := %DB23.DBB9, out1 => "DB24_AlarmDisplay".Alarm9)
   END_RUNG
   RUNG wire#w1
      { S7_GenerateENO := "TRUE" } Move(in := %DB23.DBB10, out1 => "DB24_AlarmDisplay".Alarm12)
      { S7_GenerateENO := "TRUE" } Move(in := %DB23.DBB11, out1 => "DB24_AlarmDisplay".Alarm11)
   END_RUNG
   RUNG wire#w1
      { S7_GenerateENO := "TRUE" } Move(in := %DB23.DBB12, out1 => "DB24_AlarmDisplay".Alarm14)
      { S7_GenerateENO := "TRUE" } Move(in := %DB23.DBB13, out1 => "DB24_AlarmDisplay".Alarm13)
   END_RUNG
   RUNG wire#w1
      { S7_GenerateENO := "TRUE" } Move(in := %DB23.DBB14, out1 => "DB24_AlarmDisplay".Alarm16)
      { S7_GenerateENO := "TRUE" } Move(in := %DB23.DBB15, out1 => "DB24_AlarmDisplay".Alarm15)
   END_RUNG
   RUNG wire#w1
      { S7_GenerateENO := "TRUE" } Move(in := %DB23.DBB16, out1 => "DB24_AlarmDisplay".Alarm18)
      { S7_GenerateENO := "TRUE" } Move(in := %DB23.DBB17, out1 => "DB24_AlarmDisplay".Alarm17)
   END_RUNG
   RUNG wire#w1
      { S7_GenerateENO := "TRUE" } Move(in := %DB23.DBB18, out1 => "DB24_AlarmDisplay".Alarm20)
      { S7_GenerateENO := "TRUE" } Move(in := %DB23.DBB19, out1 => "DB24_AlarmDisplay".Alarm19)
   END_RUNG
   RUNG wire#w1
      { S7_GenerateENO := "TRUE" } Move(in := %DB23.DBB20, out1 => "DB24_AlarmDisplay".Alarm22)
      { S7_GenerateENO := "TRUE" } Move(in := %DB23.DBB21, out1 => "DB24_AlarmDisplay".Alarm21)
   END_RUNG
   RUNG wire#w1
      { S7_GenerateENO := "TRUE" } Move(in := %DB23.DBB22, out1 => "DB24_AlarmDisplay".Alarm24)
      { S7_GenerateENO := "TRUE" } Move(in := %DB23.DBB23, out1 => "DB24_AlarmDisplay".Alarm23)
   END_RUNG
   RUNG wire#w1
      { S7_GenerateENO := "TRUE" } Move(in := %DB23.DBB24, out1 => "DB24_AlarmDisplay".Alarm26)
      { S7_GenerateENO := "TRUE" } Move(in := %DB23.DBB25, out1 => "DB24_AlarmDisplay".Alarm25)
   END_RUNG
   RUNG wire#w1
      { S7_GenerateENO := "TRUE" } Move(in := %DB23.DBB26, out1 => "DB24_AlarmDisplay".Alarm28)
      { S7_GenerateENO := "TRUE" } Move(in := %DB23.DBB27, out1 => "DB24_AlarmDisplay".Alarm27)
   END_RUNG
   RUNG wire#w1
      { S7_GenerateENO := "TRUE" } Move(in := %DB23.DBB28, out1 => "DB24_AlarmDisplay".Alarm30)
      { S7_GenerateENO := "TRUE" } Move(in := %DB23.DBB29, out1 => "DB24_AlarmDisplay".Alarm29)
   END_RUNG
   // the same network as SCL:
   // ENO of a box is taken as its EN; it also drops when the box reports an error
   IF "On" THEN
       "DB24_AlarmDisplay".Alarm2 := %DB23.DBB0;
       "DB24_AlarmDisplay".Alarm1 := %DB23.DBB1;
       "DB24_AlarmDisplay".Alarm4 := %DB23.DBB2;
       "DB24_AlarmDisplay".Alarm3 := %DB23.DBB3;
       "DB24_AlarmDisplay".Alarm6 := %DB23.DBB4;
       "DB24_AlarmDisplay".Alarm5 := %DB23.DBB5;
       "DB24_AlarmDisplay".Alarm8 := %DB23.DBB6;
       "DB24_AlarmDisplay".Alarm7 := %DB23.DBB7;
       "DB24_AlarmDisplay".Alarm10 := %DB23.DBB8;
       "DB24_AlarmDisplay".Alarm9 := %DB23.DBB9;
       "DB24_AlarmDisplay".Alarm12 := %DB23.DBB10;
       "DB24_AlarmDisplay".Alarm11 := %DB23.DBB11;
       "DB24_AlarmDisplay".Alarm14 := %DB23.DBB12;
       "DB24_AlarmDisplay".Alarm13 := %DB23.DBB13;
       "DB24_AlarmDisplay".Alarm16 := %DB23.DBB14;
       "DB24_AlarmDisplay".Alarm15 := %DB23.DBB15;
       "DB24_AlarmDisplay".Alarm18 := %DB23.DBB16;
       "DB24_AlarmDisplay".Alarm17 := %DB23.DBB17;
       "DB24_AlarmDisplay".Alarm20 := %DB23.DBB18;
       "DB24_AlarmDisplay".Alarm19 := %DB23.DBB19;
       "DB24_AlarmDisplay".Alarm22 := %DB23.DBB20;
       "DB24_AlarmDisplay".Alarm21 := %DB23.DBB21;
       "DB24_AlarmDisplay".Alarm24 := %DB23.DBB22;
       "DB24_AlarmDisplay".Alarm23 := %DB23.DBB23;
       "DB24_AlarmDisplay".Alarm26 := %DB23.DBB24;
       "DB24_AlarmDisplay".Alarm25 := %DB23.DBB25;
       "DB24_AlarmDisplay".Alarm28 := %DB23.DBB26;
       "DB24_AlarmDisplay".Alarm27 := %DB23.DBB27;
       "DB24_AlarmDisplay".Alarm30 := %DB23.DBB28;
       "DB24_AlarmDisplay".Alarm29 := %DB23.DBB29;
   END_IF;
END_REGION
END_FUNCTION

FUNCTION "FC41_NoRopeUnit" : Void   // FC41, LAD
TITLE = No rope unit
{ S7_Optimized_Access := 'FALSE' }
AUTHOR : Robopac
VERSION : 0.0
// stored: AutoNumber false, IsIECCheckEnabled false, SetENOAutomatically false, UDAEnableTagReadback false
BEGIN

REGION Network 1: RopeUnitOk1: Rope unit open
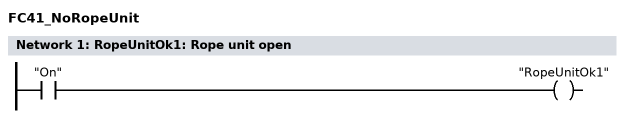
   RUNG wire#powerrail
      Contact( "On" )
      Coil( "RopeUnitOk1" )
   END_RUNG
   // the same network as SCL:
   "RopeUnitOk1" := "On";
END_REGION
END_FUNCTION

FUNCTION "FC43_PreCarriageTechnoplat" : Void   // FC43, LAD
TITLE = HS40 standard prestretch management
{ S7_Optimized_Access := 'FALSE' }
AUTHOR : Robopac
VERSION : 0.0
// stored: AutoNumber false, IsIECCheckEnabled false, SetENOAutomatically false, UDAEnableTagReadback false
BEGIN

REGION Network 1: Timer for prestretch restart
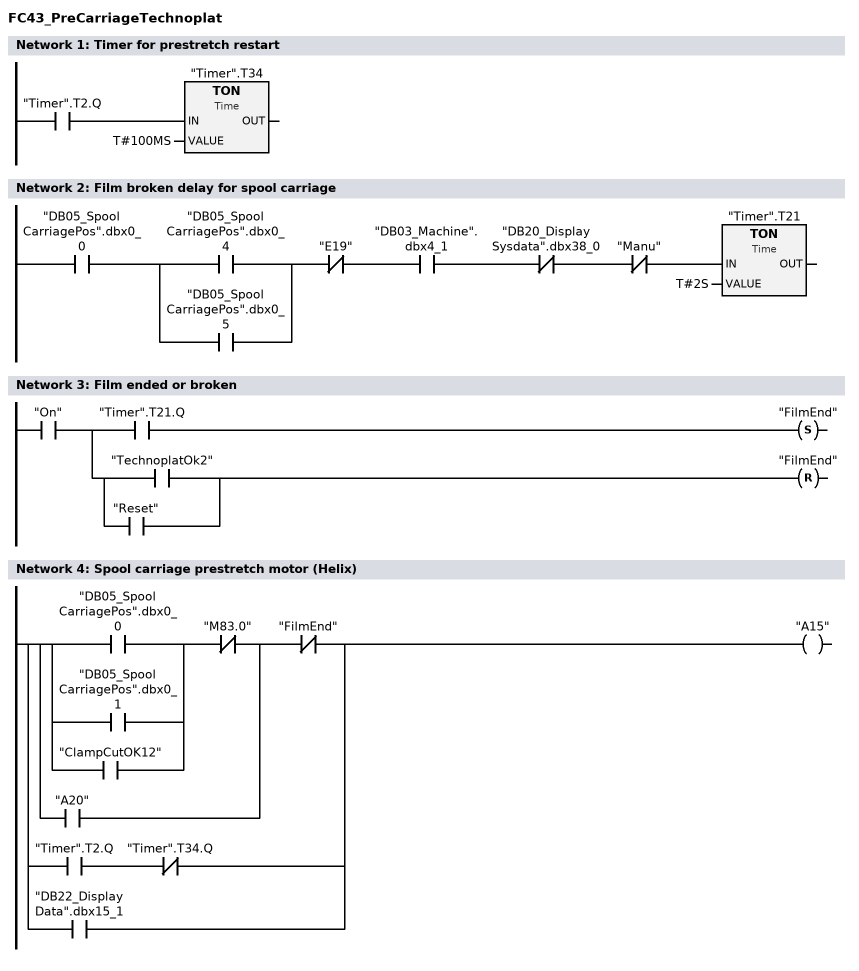
   "Timer".T34.TON(IN := "Timer".T2.Q, PT := T#100MS);   // TON coil
END_REGION

REGION Network 2: Film broken delay for spool carriage
   "Timer".T21.TON(IN := "DB05_SpoolCarriagePos".dbx0_0 AND ("DB05_SpoolCarriagePos".dbx0_4 OR "DB05_SpoolCarriagePos".dbx0_5) AND NOT "E19" AND "DB03_Machine".dbx4_1 AND NOT "DB20_DisplaySysdata".dbx38_0 AND NOT "Manu", PT := T#2S);   // TON coil
END_REGION

REGION Network 3: Film ended or broken
   RUNG wire#powerrail
      Contact( "On" )
      wire#w1
      Contact( "Timer".T21.Q )
      S_Coil( "FilmEnd" )
   END_RUNG
   RUNG wire#w1
      Contact( "TechnoplatOk2" )
      wire#w2
      R_Coil( "FilmEnd" )
   END_RUNG
   RUNG wire#w1
      Contact( "Reset" )
   END_RUNG wire#w2
   // the same network as SCL:
   IF "On" AND "Timer".T21.Q THEN "FilmEnd" := TRUE; END_IF;
   IF "On" AND ("TechnoplatOk2" OR "Reset") THEN "FilmEnd" := FALSE; END_IF;
END_REGION

REGION Network 4: Spool carriage prestretch motor (Helix)
   RUNG wire#powerrail
      Contact( "DB05_SpoolCarriagePos".dbx0_0 )
      wire#w1
      I_Contact( "M83.0" )
      wire#w2
      I_Contact( "FilmEnd" )
      wire#w3
      Coil( "A15" )
   END_RUNG
   RUNG wire#powerrail
      Contact( "DB05_SpoolCarriagePos".dbx0_1 )
   END_RUNG wire#w1
   RUNG wire#powerrail
      Contact( "ClampCutOK12" )
   END_RUNG wire#w1
   RUNG wire#powerrail
      Contact( "A20" )
   END_RUNG wire#w2
   RUNG wire#powerrail
      Contact( "Timer".T2.Q )
      I_Contact( "Timer".T34.Q )
   END_RUNG wire#w3
   RUNG wire#powerrail
      Contact( "DB22_DisplayData".dbx15_1 )
   END_RUNG wire#w3
   // the same network as SCL:
   "A15" := (((("DB05_SpoolCarriagePos".dbx0_0 OR "DB05_SpoolCarriagePos".dbx0_1 OR "ClampCutOK12") AND NOT "M83.0") OR "A20") AND NOT "FilmEnd") OR ("Timer".T2.Q AND NOT "Timer".T34.Q) OR "DB22_DisplayData".dbx15_1;
END_REGION
END_FUNCTION

FUNCTION "FC58_TableRotationPos" : Void   // FC58, LAD
{ S7_Optimized_Access := 'FALSE' }
VERSION : 0.1
// stored: AutoNumber false, IsIECCheckEnabled false, SetENOAutomatically false, UDAEnableTagReadback false
   VAR_INPUT
      PHASE : Bool;
   END_VAR
   VAR_TEMP
      TempDInt3 : DInt;
      PulseOffset : DInt;
      AC1 : Real;
      AC2 : Real;
      AC3 : Real;
      DeltaV : Real;
      DeltaVMax : Real;
      VattpiuVmin : Real;
      VmaxpiuVmin : Real;
      AC1_INT : Int;
      PulseReset : Bool;
      TEMPOMAX : Real;
      TEMPO : Real;
      Encoder : Int;
      TempDint : DInt;
      TempInt : Int;
      TempDint2 : DInt;
      TempDInt4 : DInt;
      TempWord : Word;
   END_VAR
   VAR_TEMP   // added for the SCL form of the ladder/FBD networks
      _w1 : Bool;
   END_VAR
BEGIN

REGION Network 1
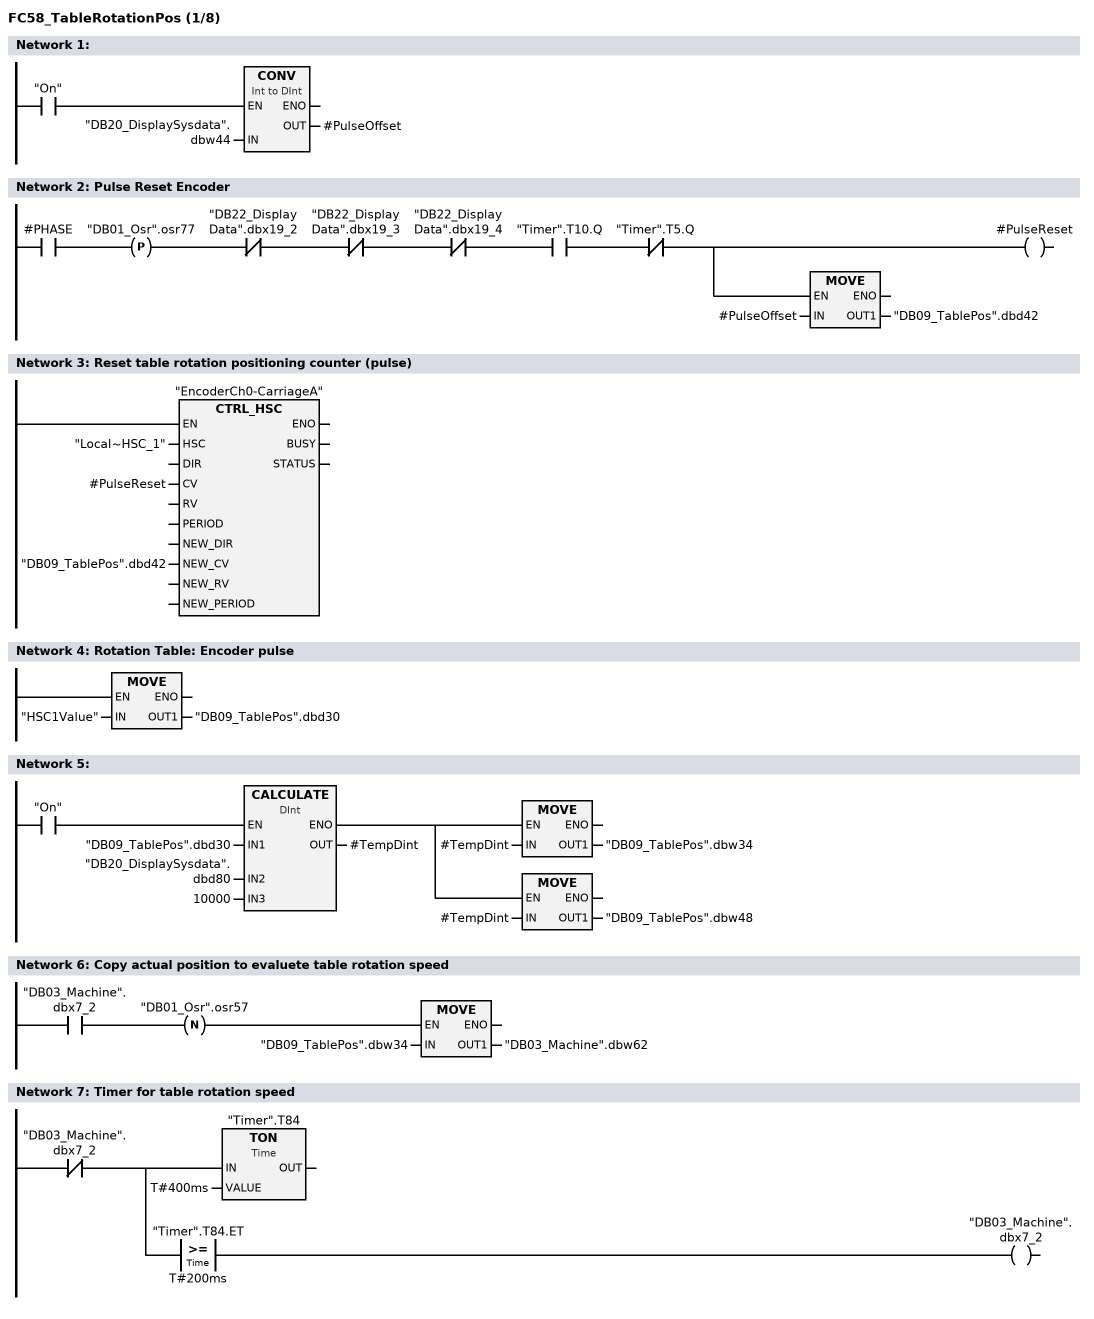
   RUNG wire#powerrail
      Contact( "On" )
      { S7_Templates := "[SrcType := Int, DestType := DInt]"; S7_GenerateENO := "TRUE" } Convert(in := "DB20_DisplaySysdata".dbw44, out => #PulseOffset)
   END_RUNG
   // the same network as SCL:
   IF "On" THEN #PulseOffset := INT_TO_DINT("DB20_DisplaySysdata".dbw44); END_IF;
END_REGION

REGION Network 2: Pulse Reset Encoder
   RUNG wire#powerrail
      Contact( #PHASE )
      P_Trig( "DB01_Osr".osr77 )
      I_Contact( "DB22_DisplayData".dbx19_2 )
      I_Contact( "DB22_DisplayData".dbx19_3 )
      I_Contact( "DB22_DisplayData".dbx19_4 )
      Contact( "Timer".T10.Q )
      I_Contact( "Timer".T5.Q )
      wire#w1
      Coil( #PulseReset )
   END_RUNG
   RUNG wire#w1
      { S7_GenerateENO := "TRUE" } Move(in := #PulseOffset, out1 => "DB09_TablePos".dbd42)
   END_RUNG
   // the same network as SCL:
   #_w1 := #PHASE AND NOT "DB01_Osr".osr77;   // rising edge
   "DB01_Osr".osr77 := #PHASE;
   #PulseReset := #_w1 AND NOT "DB22_DisplayData".dbx19_2 AND NOT "DB22_DisplayData".dbx19_3 AND NOT "DB22_DisplayData".dbx19_4 AND "Timer".T10.Q AND NOT "Timer".T5.Q;
   IF #PulseReset THEN "DB09_TablePos".dbd42 := #PulseOffset; END_IF;
END_REGION

REGION Network 3: Reset table rotation positioning counter (pulse)
   RUNG wire#powerrail
      "EncoderCh0-CarriageA".CTRL_HSC(HSC := "Local~HSC_1", DIR :=, CV := #PulseReset, RV :=, PERIOD :=, NEW_DIR :=, NEW_CV := "DB09_TablePos".dbd42, NEW_RV :=, NEW_PERIOD :=, BUSY =>, STATUS =>)
   END_RUNG
   // the same network as SCL:
   "EncoderCh0-CarriageA"(HSC := "Local~HSC_1", CV := #PulseReset, NEW_CV := "DB09_TablePos".dbd42);   // CTRL_HSC
END_REGION

REGION Network 4: Rotation Table: Encoder pulse
   RUNG wire#powerrail
      { S7_GenerateENO := "TRUE" } Move(in := "HSC1Value", out1 => "DB09_TablePos".dbd30)
   END_RUNG
   // the same network as SCL:
   "DB09_TablePos".dbd30 := "HSC1Value";
END_REGION

REGION Network 5
   RUNG wire#powerrail
      Contact( "On" )
      { S7_Templates := "SrcType := DInt"; S7_GenerateENO := "TRUE"; S7_Expression := "((In1*In2)/In3)" } Calculate(in1 := "DB09_TablePos".dbd30, in2 := "DB20_DisplaySysdata".dbd80, in3 := 10000, out => #TempDint)
      wire#w1
      { S7_GenerateENO := "TRUE" } Move(in := #TempDint, out1 => "DB09_TablePos".dbw34)
   END_RUNG
   RUNG wire#w1
      { S7_GenerateENO := "TRUE" } Move(in := #TempDint, out1 => "DB09_TablePos".dbw48)
   END_RUNG
   // the same network as SCL:
   // ENO of a box is taken as its EN; it also drops when the box reports an error
   IF "On" THEN
       #TempDint := (("DB09_TablePos".dbd30*"DB20_DisplaySysdata".dbd80)/10000);
       "DB09_TablePos".dbw34 := #TempDint;
       "DB09_TablePos".dbw48 := #TempDint;
   END_IF;
END_REGION

REGION Network 6: Copy actual position to evaluete table rotation speed
   RUNG wire#powerrail
      Contact( "DB03_Machine".dbx7_2 )
      N_Trig( "DB01_Osr".osr57 )
      { S7_GenerateENO := "TRUE" } Move(in := "DB09_TablePos".dbw34, out1 => "DB03_Machine".dbw62)
   END_RUNG
   // the same network as SCL:
   #_w1 := NOT "DB03_Machine".dbx7_2 AND "DB01_Osr".osr57;   // falling edge
   "DB01_Osr".osr57 := "DB03_Machine".dbx7_2;
   IF #_w1 THEN "DB03_Machine".dbw62 := "DB09_TablePos".dbw34; END_IF;
END_REGION

REGION Network 7: Timer for table rotation speed
   #_w1 := NOT "DB03_Machine".dbx7_2;
   "Timer".T84.TON(IN := #_w1, PT := T#400ms);   // TON coil
   "DB03_Machine".dbx7_2 := #_w1 AND ("Timer".T84.ET >= T#200ms);
END_REGION

REGION Network 8: Speed calculation (1)
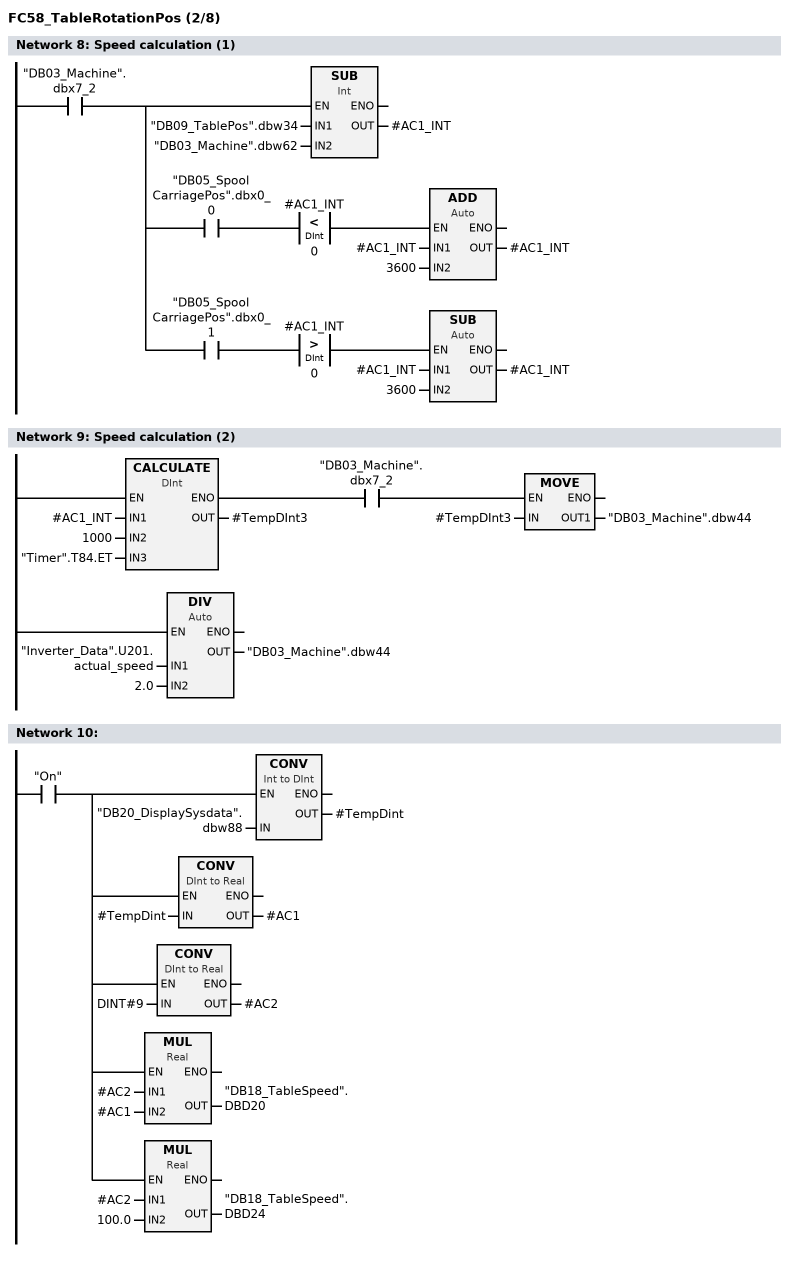
   RUNG wire#powerrail
      Contact( "DB03_Machine".dbx7_2 )
      wire#w1
      { S7_Templates := "SrcType := Int"; S7_GenerateENO := "TRUE" } Sub(in1 := "DB09_TablePos".dbw34, in2 := "DB03_Machine".dbw62, out => #AC1_INT)
   END_RUNG
   RUNG wire#w1
      Contact( "DB05_SpoolCarriagePos".dbx0_0 )
      { S7_Templates := "SrcType := DInt" } LT_Contact(in1 := #AC1_INT, in2 := 0)
      { S7_GenerateENO := "TRUE" } Add(in1 := #AC1_INT, in2 := 3600, out => #AC1_INT)
   END_RUNG
   RUNG wire#w1
      Contact( "DB05_SpoolCarriagePos".dbx0_1 )
      { S7_Templates := "SrcType := DInt" } GT_Contact(in1 := #AC1_INT, in2 := 0)
      { S7_GenerateENO := "TRUE" } Sub(in1 := #AC1_INT, in2 := 3600, out => #AC1_INT)
   END_RUNG
   // the same network as SCL:
   IF "DB03_Machine".dbx7_2 THEN #AC1_INT := "DB09_TablePos".dbw34 - "DB03_Machine".dbw62; END_IF;
   IF "DB03_Machine".dbx7_2 AND "DB05_SpoolCarriagePos".dbx0_0 AND (#AC1_INT < 0) THEN
       #AC1_INT := #AC1_INT + 3600;
   END_IF;
   IF "DB03_Machine".dbx7_2 AND "DB05_SpoolCarriagePos".dbx0_1 AND (#AC1_INT > 0) THEN
       #AC1_INT := #AC1_INT - 3600;
   END_IF;
END_REGION

REGION Network 9: Speed calculation (2)
   RUNG wire#powerrail
      { S7_Templates := "SrcType := DInt"; S7_GenerateENO := "TRUE"; S7_Expression := "((In1*In2)/In3)" } Calculate(in1 := #AC1_INT, in2 := 1000, in3 := "Timer".T84.ET, out => #TempDInt3)
      Contact( "DB03_Machine".dbx7_2 )
      { S7_GenerateENO := "TRUE" } Move(in := #TempDInt3, out1 => "DB03_Machine".dbw44)
   END_RUNG
   RUNG wire#powerrail
      Div(in1 := "Inverter_Data".U201.actual_speed, in2 := 2.0, out => "DB03_Machine".dbw44)
   END_RUNG
   // the same network as SCL:
   // ENO of a box is taken as its EN; it also drops when the box reports an error
   #TempDInt3 := ((#AC1_INT*1000)/"Timer".T84.ET);
   IF "DB03_Machine".dbx7_2 THEN "DB03_Machine".dbw44 := #TempDInt3; END_IF;
   "DB03_Machine".dbw44 := "Inverter_Data".U201.actual_speed / 2.0;
END_REGION

REGION Network 10
   RUNG wire#powerrail
      Contact( "On" )
      wire#w1
      { S7_Templates := "[SrcType := Int, DestType := DInt]"; S7_GenerateENO := "TRUE" } Convert(in := "DB20_DisplaySysdata".dbw88, out => #TempDint)
   END_RUNG
   RUNG wire#w1
      { S7_Templates := "[SrcType := DInt, DestType := Real]"; S7_GenerateENO := "TRUE" } Convert(in := #TempDint, out => #AC1)
   END_RUNG
   RUNG wire#w1
      { S7_Templates := "[SrcType := DInt, DestType := Real]"; S7_GenerateENO := "TRUE" } Convert(in := DINT#9, out => #AC2)
   END_RUNG
   RUNG wire#w1
      { S7_Templates := "SrcType := Real"; S7_GenerateENO := "TRUE" } Mul(in1 := #AC2, in2 := #AC1, out => "DB18_TableSpeed".DBD20)
   END_RUNG
   RUNG wire#w1
      { S7_Templates := "SrcType := Real"; S7_GenerateENO := "TRUE" } Mul(in1 := #AC2, in2 := 100.0, out => "DB18_TableSpeed".DBD24)
   END_RUNG
   // the same network as SCL:
   IF "On" THEN
       #TempDint := INT_TO_DINT("DB20_DisplaySysdata".dbw88);
       #AC1 := DINT_TO_REAL(#TempDint);
       #AC2 := DINT_TO_REAL(DINT#9);
       "DB18_TableSpeed".DBD20 := #AC2 * #AC1;
       "DB18_TableSpeed".DBD24 := #AC2 * 100.0;
   END_IF;
END_REGION

REGION Network 11
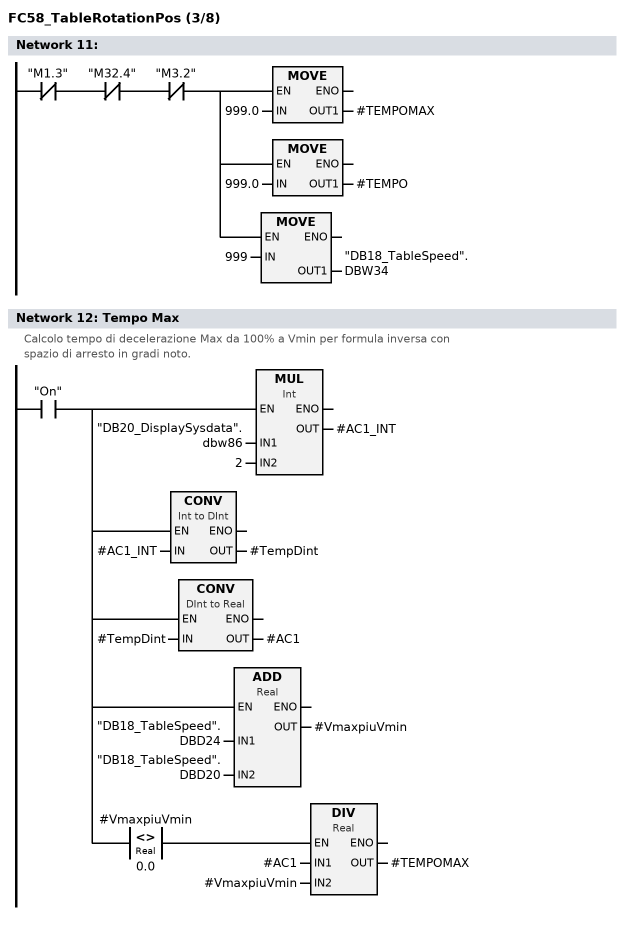
   RUNG wire#powerrail
      I_Contact( "M1.3" )
      I_Contact( "M32.4" )
      I_Contact( "M3.2" )
      wire#w1
      { S7_GenerateENO := "TRUE" } Move(in := 999.0, out1 => #TEMPOMAX)
   END_RUNG
   RUNG wire#w1
      { S7_GenerateENO := "TRUE" } Move(in := 999.0, out1 => #TEMPO)
   END_RUNG
   RUNG wire#w1
      { S7_GenerateENO := "TRUE" } Move(in := 999, out1 => "DB18_TableSpeed".DBW34)
   END_RUNG
   // the same network as SCL:
   IF NOT "M1.3" AND NOT "M32.4" AND NOT "M3.2" THEN
       #TEMPOMAX := 999.0;
       #TEMPO := 999.0;
       "DB18_TableSpeed".DBW34 := 999;
   END_IF;
END_REGION

REGION Network 12: Tempo Max
   // Calcolo tempo di decelerazione Max da 100% a Vmin per formula inversa con 
   // spazio di arresto in gradi noto.
   RUNG wire#powerrail
      Contact( "On" )
      wire#w1
      { S7_Templates := "SrcType := Int"; S7_GenerateENO := "TRUE" } Mul(in1 := "DB20_DisplaySysdata".dbw86, in2 := 2, out => #AC1_INT)
   END_RUNG
   RUNG wire#w1
      { S7_Templates := "[SrcType := Int, DestType := DInt]"; S7_GenerateENO := "TRUE" } Convert(in := #AC1_INT, out => #TempDint)
   END_RUNG
   RUNG wire#w1
      { S7_Templates := "[SrcType := DInt, DestType := Real]"; S7_GenerateENO := "TRUE" } Convert(in := #TempDint, out => #AC1)
   END_RUNG
   RUNG wire#w1
      { S7_Templates := "SrcType := Real"; S7_GenerateENO := "TRUE" } Add(in1 := "DB18_TableSpeed".DBD24, in2 := "DB18_TableSpeed".DBD20, out => #VmaxpiuVmin)
   END_RUNG
   RUNG wire#w1
      { S7_Templates := "SrcType := Real" } NE_Contact(in1 := #VmaxpiuVmin, in2 := 0.0)
      { S7_Templates := "SrcType := Real"; S7_GenerateENO := "TRUE" } Div(in1 := #AC1, in2 := #VmaxpiuVmin, out => #TEMPOMAX)
   END_RUNG
   // the same network as SCL:
   IF "On" THEN
       #AC1_INT := "DB20_DisplaySysdata".dbw86 * 2;
       #TempDint := INT_TO_DINT(#AC1_INT);
       #AC1 := DINT_TO_REAL(#TempDint);
       #VmaxpiuVmin := "DB18_TableSpeed".DBD24 + "DB18_TableSpeed".DBD20;
   END_IF;
   IF "On" AND (#VmaxpiuVmin <> 0.0) THEN #TEMPOMAX := #AC1 / #VmaxpiuVmin; END_IF;
END_REGION

REGION Network 13: Calcolo tempo di decelerazione da Vatt a Vmin per calcolo spazio di arresto
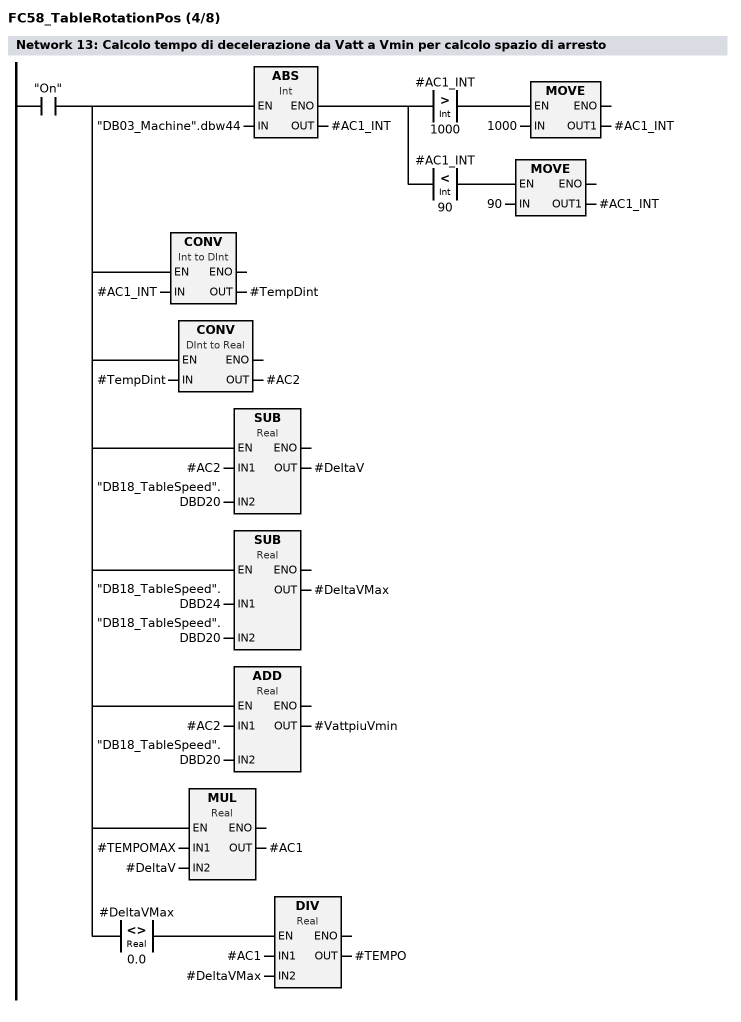
   RUNG wire#powerrail
      Contact( "On" )
      wire#w1
      { S7_Templates := "SrcType := Int" } Abs(in := "DB03_Machine".dbw44, out => #AC1_INT)
      wire#w2
      { S7_Templates := "SrcType := Int" } GT_Contact(in1 := #AC1_INT, in2 := 1000)
      Move(in := 1000, out1 => #AC1_INT)
   END_RUNG
   RUNG wire#w2
      { S7_Templates := "SrcType := Int" } LT_Contact(in1 := #AC1_INT, in2 := 90)
      Move(in := 90, out1 => #AC1_INT)
   END_RUNG
   RUNG wire#w1
      { S7_Templates := "[SrcType := Int, DestType := DInt]"; S7_GenerateENO := "TRUE" } Convert(in := #AC1_INT, out => #TempDint)
   END_RUNG
   RUNG wire#w1
      { S7_Templates := "[SrcType := DInt, DestType := Real]"; S7_GenerateENO := "TRUE" } Convert(in := #TempDint, out => #AC2)
   END_RUNG
   RUNG wire#w1
      { S7_Templates := "SrcType := Real"; S7_GenerateENO := "TRUE" } Sub(in1 := #AC2, in2 := "DB18_TableSpeed".DBD20, out => #DeltaV)
   END_RUNG
   RUNG wire#w1
      { S7_Templates := "SrcType := Real"; S7_GenerateENO := "TRUE" } Sub(in1 := "DB18_TableSpeed".DBD24, in2 := "DB18_TableSpeed".DBD20, out => #DeltaVMax)
   END_RUNG
   RUNG wire#w1
      { S7_Templates := "SrcType := Real"; S7_GenerateENO := "TRUE" } Add(in1 := #AC2, in2 := "DB18_TableSpeed".DBD20, out => #VattpiuVmin)
   END_RUNG
   RUNG wire#w1
      { S7_Templates := "SrcType := Real"; S7_GenerateENO := "TRUE" } Mul(in1 := #TEMPOMAX, in2 := #DeltaV, out => #AC1)
   END_RUNG
   RUNG wire#w1
      { S7_Templates := "SrcType := Real" } NE_Contact(in1 := #DeltaVMax, in2 := 0.0)
      { S7_Templates := "SrcType := Real"; S7_GenerateENO := "TRUE" } Div(in1 := #AC1, in2 := #DeltaVMax, out => #TEMPO)
   END_RUNG
   // the same network as SCL:
   IF "On" THEN #AC1_INT := ABS("DB03_Machine".dbw44); END_IF;
   IF "On" AND (#AC1_INT > 1000) THEN #AC1_INT := 1000; END_IF;
   IF "On" AND (#AC1_INT < 90) THEN #AC1_INT := 90; END_IF;
   IF "On" THEN
       #TempDint := INT_TO_DINT(#AC1_INT);
       #AC2 := DINT_TO_REAL(#TempDint);
       #DeltaV := #AC2 - "DB18_TableSpeed".DBD20;
       #DeltaVMax := "DB18_TableSpeed".DBD24 - "DB18_TableSpeed".DBD20;
       #VattpiuVmin := #AC2 + "DB18_TableSpeed".DBD20;
       #AC1 := #TEMPOMAX * #DeltaV;
   END_IF;
   IF "On" AND (#DeltaVMax <> 0.0) THEN #TEMPO := #AC1 / #DeltaVMax; END_IF;
END_REGION

REGION Network 14: Decelerazione
